// TwinCAT 3 PLC project PLC
// ProgramVersion: 3.1.4026.20
// libraries:
//   Tc2_Standard, * (Beckhoff Automation GmbH)
//   Tc2_System, * (Beckhoff Automation GmbH)
//   Tc2_Utilities, * (Beckhoff Automation GmbH)
//   Tc3_EventLogger, * (Beckhoff Automation GmbH)
// project tree:
//   DUTs/HMI/ ST_Batch_HMI.TcDUT, ST_Camera_HMI.TcDUT, ST_Counter_HMI.TcDUT, ST_Feeder_HMI.TcDUT, ST_Footer_HMI.TcDUT, ST_FromHMI.TcDUT, ST_Greasing_HMI.TcDUT, ST_History_HMI.TcDUT, ST_Lift_HMI.TcDUT, ST_MachineControl_HMI.TcDUT, ST_MachineInfo_HMI.TcDUT, ST_Navigation_HMI.TcDUT, ST_PID_HMI.TcDUT, ST_Robot_HMI.TcDUT, ST_Station_HMI.TcDUT, ST_ToHMI.TcDUT
//   DUTs/ ST_Alarm.TcDUT, ST_Batch.TcDUT, ST_Control.TcDUT, ST_Settings.TcDUT, ST_StationCommand.TcDUT
//   DUTs/Time/ ST_DateAndTime.TcDUT, ST_Time.TcDUT
//   DUTs/Trend/ ST_Point.TcDUT
//   FBs/Devices/ FB_Counter.TcPOU, FB_Device.TcPOU, FB_Greaser.TcPOU, FB_Handshake.TcPOU, FB_Stepper.TcPOU
//   FBs/ FB_AlarmDiagnostic.TcPOU, FB_Batch.TcPOU, FB_SystemDateTime.TcPOU, FB_TONP.TcPOU
//   Functions/ F_Message.TcPOU, F_StepCMP.TcPOU, F_TimerToString.TcPOU
//   GVLs/ CONST.TcGVL, GV.TcGVL, HMI.TcGVL, IN.TcGVL, OUT.TcGVL, Station.TcGVL
//   / PlcTask.TcTTO
//   POUs/ MAIN.TcPOU, P00_Mapping.TcPOU, P01_AnalogScaling.TcPOU, P02_GlobalSystemTime.TcPOU, P03_MachineControl.TcPOU, P05_DeviceControl.TcPOU, P06_ProcessControl.TcPOU, P99_HMIControl.TcPOU
//   POUs/Sequences/ Camera.TcPOU, Conveyor.TcPOU, Feeder.TcPOU, Greaser.TcPOU, IntakeBuffer.TcPOU, OutletBuffer.TcPOU, Robot.TcPOU
//   POUs/Simulation/ Service_sim.TcPOU, Simulation.TcPOU
// real-time tasks:
//   TASK PlcTask: cycle T#10ms, priority 20, ADS port 350

CONFIGURATION PLC
    RESOURCE PLC ON TwinCAT3
        TASK PlcTask(INTERVAL := T#10ms, PRIORITY := 20);
        PROGRAM MAIN WITH PlcTask : MAIN;
    END_RESOURCE
END_CONFIGURATION

// ---- DUTs/HMI/ST_Batch_HMI.TcDUT
TYPE ST_Batch_HMI :
STRUCT
	bBatchOpen : BOOL;
	bBatchClose : BOOL;
	sBatchName : STRING;
END_STRUCT
END_TYPE

// ---- DUTs/HMI/ST_Camera_HMI.TcDUT
TYPE ST_Camera_HMI :
STRUCT
	bCapturing		:BOOL;
	sCameraStatus	:STRING;
	sJobResult		:STRING;
END_STRUCT
END_TYPE

// ---- DUTs/HMI/ST_Counter_HMI.TcDUT
TYPE ST_Counter_HMI :
STRUCT
	bReset			:BOOL;
	iOK				:UDINT;
	iNOK			:UDINT;
	bError			:BOOL;
END_STRUCT
END_TYPE

// ---- DUTs/HMI/ST_Feeder_HMI.TcDUT
TYPE ST_Feeder_HMI :
STRUCT
	bActivate		:BOOL;
	bDeactivate		:BOOL;
END_STRUCT
END_TYPE

// ---- DUTs/HMI/ST_Footer_HMI.TcDUT
TYPE ST_Footer_HMI :
STRUCT
	bAuto : BOOL; 
	bService : BOOL;
	bStop : BOOL;
	bStart : BOOL;
	bPause : BOOL;
	
	bAuto_Enable : BOOL;
	bService_Enable : BOOL;
	bStop_Enable : BOOL;
	bStart_Enable : BOOL;
	bPause_Enable : BOOL;
END_STRUCT
END_TYPE

// ---- DUTs/HMI/ST_FromHMI.TcDUT
TYPE ST_FromHMI :
STRUCT
	stMachineCtrl		: ST_MachineControl_HMI; //Footer commands
	stNavigation		: ST_Navigation_HMI;
	stRobot				: ST_Robot_HMI;
	stLiftIntake		: ST_Lift_HMI;
	stLiftOutlet		: ST_Lift_HMI;
	bConveyorJog		: BOOL;
	bRobotCameraCapture	: BOOL;
	bFixedCameraCapture	: BOOL;
	stBatch				: ST_Batch_HMI;
	stCounter			:ARRAY [1..4] OF ST_Counter_HMI;
	stGreasing			: ST_Greasing_HMI;
	iSelectedTray		: USINT;
	stFeeder			:ST_Feeder_HMI;
END_STRUCT
END_TYPE

// ---- DUTs/HMI/ST_Greasing_HMI.TcDUT
TYPE ST_Greasing_HMI :
STRUCT
	bPurge		:BOOL;
	bPulse		:BOOL;
	iTime		:UINT;
END_STRUCT
END_TYPE

// ---- DUTs/HMI/ST_History_HMI.TcDUT
TYPE ST_History_HMI :
STRUCT
	iOK	:UDINT;
	iNOK :UDINT;
	bShift1	:BOOL;
	bShift2 :BOOL;
	bShift3 :BOOL;
END_STRUCT
END_TYPE

// ---- DUTs/HMI/ST_Lift_HMI.TcDUT
TYPE ST_Lift_HMI :
STRUCT
	bHome		:BOOL;
	bGoUp		:BOOL;
	bGoDown		:BOOL;
	iPosition	:UINT;
END_STRUCT
END_TYPE

// ---- DUTs/HMI/ST_MachineControl_HMI.TcDUT
TYPE ST_MachineControl_HMI :
STRUCT
	bAutomaticMode 		: BOOL;
	bServiceMode		: BOOL;
	
	bStartProcess		: BOOL;
	bPauseProcess		: BOOL;
	bStopProcess		: BOOL;
	
	
END_STRUCT
END_TYPE

// ---- DUTs/HMI/ST_MachineInfo_HMI.TcDUT
TYPE ST_MachineInfo_HMI :
STRUCT
	bControlMode		: BOOL;//0 - Auto, 1 - Manual
	iStatus				: USINT;//0-Stopping, 1-Stopped, 2-Starting, 3-Running, 4-Paused
	sBatch				: STRING;// Closed or Batch number
	iCounter			: LINT;//Finished part counter
	sDate				: STRING;//System date
	sTime				: STRING;//System time
	sCycleTime			: STRING;//MM:SS
	sUserLogged			: STRING;
	iCurrentStep		: USINT;
	
END_STRUCT
END_TYPE

// ---- DUTs/HMI/ST_Navigation_HMI.TcDUT
TYPE ST_Navigation_HMI :
STRUCT
	
END_STRUCT
END_TYPE

// ---- DUTs/HMI/ST_PID_HMI.TcDUT
TYPE ST_PID_HMI :
STRUCT
	bTray_PickPosition	: BOOL;
	bTray_PlacePosition	: BOOL;
	bTray_Ready_Left	: BOOL;
	bTray_Ready_Right	: BOOL;
	bConveyor_Moving	: BOOL;
END_STRUCT
END_TYPE

// ---- DUTs/HMI/ST_Robot_HMI.TcDUT
TYPE ST_Robot_HMI :
STRUCT
	bStart : BOOL;
	bStop : BOOL;
	bInit : BOOL;
	bPause	: BOOL;
	bPowerOn : BOOL;
	bPowerOff : BOOL;
	
	iStep : 	UINT;
	sStatus : STRING;
END_STRUCT
END_TYPE

// ---- DUTs/HMI/ST_Station_HMI.TcDUT
TYPE ST_Station_HMI :
STRUCT
	iStep			:UINT;
	bInterlocksOK	:BOOL;
	bReset			:BOOL;
	iStatus			:UINT;
END_STRUCT
END_TYPE

// ---- DUTs/HMI/ST_ToHMI.TcDUT
TYPE ST_ToHMI :
STRUCT
	stHeader		:ST_MachineInfo_HMI;
	stPID			:ST_PID_HMI;
	stFooter		:ST_Footer_HMI;
	stRobot			:ST_Robot_HMI;
	stLiftIntake	:ST_Lift_HMI;
	stLiftOutlet	:ST_Lift_HMI;
	bConveyorJog	:BOOL;
	stRobotCamera	:ST_Camera_HMI;
	stFixedCamera	:ST_Camera_HMI;
	stBatch			:ST_Batch_HMI;
	stCounter		:ARRAY [1..7] OF ST_Counter_HMI;
	stGreasing		:ST_Greasing_HMI;
	stHistory		:ST_History_HMI;
	iMessage		:UINT;
	iMessageSeverity :USINT;
	stFeeder		:ST_Feeder_HMI;
END_STRUCT
END_TYPE

// ---- DUTs/ST_Alarm.TcDUT
TYPE ST_Alarm :
STRUCT
	Alarm			:ARRAY[0..50] OF fb_TcAlarm;
	Active			:ARRAY[0..50] OF BOOL;
	Raise			:ARRAY[0..50] OF BOOL;
	
END_STRUCT
END_TYPE

// ---- DUTs/ST_Batch.TcDUT
TYPE ST_Batch :
STRUCT
	sBatchNumber		:STRING;
	sRecipeName			:STRING;
	sProductName		:STRING;
	sUser				:STRING;
	sStarted			:STRING;
	sFinished			:STRING;
END_STRUCT
END_TYPE

// ---- DUTs/ST_Control.TcDUT
TYPE ST_Control :
STRUCT
	iStep					:UINT;
	iStep_Prev				:UINT;
	bAuto					:BOOL;
	bService				:BOOL;
	bStarting				:BOOL;
	bInterlockOK			:BOOL;
	bProcesslockOK			:BOOL;
	bStartConditionsOK		:BOOL;
	bRunning				:BOOL;
	bPaused					:BOOL;
	bAbort					:BOOL;
	bStopping				:BOOL;
	bStopped				:BOOL;
	bJump					:BOOL;
	bHold					:BOOL;
	bPoweredOn				:BOOL;
	bPoweredOff				:BOOL;
	bInit					:BOOL;
END_STRUCT
END_TYPE

// ---- DUTs/ST_Settings.TcDUT
TYPE ST_Settings :
STRUCT
	//Timeout settings
	tCameraTimeout			:TIME;
	tConveyorTimeout		:TIME;
	tPickClampTimeout		:TIME;
	tPlaceClampTimeout		:TIME;
	tFeederTimeout			:TIME;
	tRobotTimeout			:TIME;
	
	//Process settings
	tGreasingPulseTime		:TIME;
END_STRUCT
END_TYPE

// ---- DUTs/ST_StationCommand.TcDUT
TYPE ST_StationCommand :
STRUCT
	//Feeder cmd
	bFeederSTART		:BOOL;
	//Intake lift cmd
	iIntakeLift_SP		:UINT;
	bIntakeLift_HOME	:BOOL;
	//Outlet lift cmd
	iOutletLift_SP		:UINT;
	bOutletLift_HOME	:BOOL;
	//Robot cmd
	bRobot_START		:BOOL;
	iRobot_JobNumber	:USINT;
	bRobot_Gripper		:BYTE;
	//Conveyor cmd
	bConveyorJog		:BOOL;
	bClampPick			:BOOL;
	bClampPlace			:BOOL;
	//Robot camera cmd
	bRobotCamera_Capture:BOOL;
	//Fixed camera cmd
	bFixedCamera_Capture:BOOL;
	iFixedCamera_Job	:USINT;
	//Counters
	bCount				:BOOL;
	iPartOK				:USINT;
	iPartNOK			:USINT;
	//Greasing
	bGreasing_Purge		:BOOL;
	bGreasing_Pulse		:BOOL;
	tGreasing_Time		:TIME;
END_STRUCT
END_TYPE

// ---- DUTs/Time/ST_DateAndTime.TcDUT
TYPE ST_DateAndTime :
STRUCT
END_STRUCT
END_TYPE

// ---- DUTs/Time/ST_Time.TcDUT
TYPE ST_Time :
STRUCT
	dtDateTime			:DT;
	sTime				:STRING;
	sDate				:STRING;
	sDateTime			:STRING;
	sFormatDateTime		:STRING;
	bClock_500ms		:BOOL;
	bClock_1s			:BOOL;
	bClock_2s			:BOOL;
	bClock_5s			:BOOL;
	bClock_60s			:BOOL;
	bClock_1OFF_2ON		:BOOL;
	bPulse_10s			:BOOL;
	bPulse_30s			:BOOL;
	bPulse_60s			:BOOL;
	bCustomBlink1		:BOOL;
	bCustomBlink2		:BOOL;
	bCustomBlink3		:BOOL;
	bNewHour			:BOOL;
	bNewDay				:BOOL;
	bNewMonth			:BOOL;
	bNewYear			:BOOL;
	CurrentHour			:WORD;
	CurrentDay			:WORD;
	CurrentMonth		:WORD;
	CurrentYear			:WORD;
END_STRUCT
END_TYPE

// ---- DUTs/Trend/ST_Point.TcDUT
TYPE ST_Point :
STRUCT
	x	:UDINT;
	y	:UDINT;
END_STRUCT
END_TYPE

// ---- GVLs/CONST.TcGVL
{attribute 'qualified_only'}
VAR_GLOBAL
	AMS_NETID				:STRING:='10.0.0.5.1.1';
	PROJECT_DIR				:STRING:='C:\250605-Aeromatic1\';
	DB_ID					:UDINT:=1;
	
	
	//Process constants
	GREASE_DENSITY			:REAL:=1;//[g/l]
	
	
	//Message IDs
	MSG_FillIntakeBuffer	:UINT := 10;
	
END_VAR

// ---- GVLs/GV.TcGVL
{attribute 'qualified_only'}
VAR_GLOBAL
	//Time
	stTime : ST_Time;
	bUPSDetect : BOOL;
END_VAR

VAR_GLOBAL PERSISTENT
	sUserLogged					:STRING;
	cntResettable				:FB_Counter;
	cntHourly					:FB_Counter;
	cntTotal					:FB_Counter;
	cntBatch					:FB_Counter;
	cntShift1					:FB_Counter;
	cntShift2					:FB_Counter;
	cntShift3					:FB_Counter;
	stSettings					:ST_Settings;
	aTrays						:ARRAY[1..10] OF ARRAY[1..14,1..7] OF BOOL;
END_VAR

// ---- GVLs/HMI.TcGVL
{attribute 'qualified_only'}
VAR_GLOBAL
	stToHMI 			:ST_ToHMI;
	stFromHMI 			:ST_FromHMI; 
	iMenu 				:USINT;
	iPopupMenu 			:USINT;
	stGreasing			:ST_Station_HMI;
	stInletBuffer		:ST_Station_HMI;
	stOutletBuffer		:ST_Station_HMI;
	stConveyor			:ST_Station_HMI;
	stRobot				:ST_Station_HMI;
	stCamera			:ST_Station_HMI;
	stFeeder			:ST_Station_HMI;
	stLastTray			:ARRAY[1..14,1..7] OF BOOL;
END_VAR

// ---- GVLs/IN.TcGVL
{attribute 'qualified_only'}
VAR_GLOBAL
	//Input modules:


	//Input variables:	
	
	//Sensors
	bSensor_TrayInReady		:BOOL;
	bSensor_TrayOutReady	:BOOL;
	bSensor_TrayInPick		:BOOL;
	bSensor_TrayInPlace		:BOOL;
	bSensor_InletDoor_Closed	:BOOL;
	bSensor_OutletDoor_Closed	:BOOL;
	
	//Robot
	bRobot_Initialised		:BOOL;
	bRobot_Running			:BOOL;
	bRobot_Ready			:BOOL;
	bRobot_On				:BOOL;
	bRobot_Ok				:BOOL;
	bRobot_Done				:BOOL;
	bRobot_Gripper			:BYTE;
	bRobot_Args				:BYTE;
	
	//Camera
	bCamera_Busy			:BOOL;
	bCamera_Done			:BOOL;
	bCamera_Args			:BYTE;
	bCamera_On				:BOOL;
	
	//Conveyor
	bConveyor_Drive			:BOOL;
	bPickClamped			:BOOL;
	bPlaceClamped			:BOOL;
	bConveyorDrive_OK		:BOOL;
	
	//Feeder
	bFeeder_ON				:BOOL;
	bFeederDrive_OK			:BOOL;
	
	//Intake buffer
	bIntakeBuffer_Homed		:BOOL;
	iBufferIn				:INT;
	bIntakeBuffer_DriveOK	:BOOL;
	//Outlet buffer
	bOutletBuffer_Homed		:BOOL;
	iBufferOut				:INT;
	bOutletBuffer_DriveOK	:BOOL;
	
	//Greaser
	bGreasing_PressureOK	:BOOL;
	bGreasing_LevelOK		:BOOL;

END_VAR

// ---- GVLs/OUT.TcGVL
{attribute 'qualified_only'}
VAR_GLOBAL
	//Camera
	bFixedCamera_Trigger		:BOOL;
	FixedCameraArgs				:ARRAY[0..9] OF BOOL;
	bFixedCamera_PlcReady		:BOOL;
	//Conveyor
	bConveyor_Jog				:BOOL;
	bClampPick					:BOOL;
	bClampPlace					:BOOL;
	//Robot
	bRobot_Execute				:BOOL;
	bRobot_PlcReady				:BOOL;
END_VAR

// ---- GVLs/Station.TcGVL
{attribute 'qualified_only'}
VAR_GLOBAL
	stAlarm							:ST_Alarm;

	bBatchOpen						:BOOL;
	bBatchClosed						:BOOL;
	bBatchBusy						:BOOL;
	bAlarmOK						:BOOL;	
	
	stAutoCmd						:ST_StationCommand;
	stManCmd						:ST_StationCommand;
	stCommand						:ST_StationCommand;				

	tonCycleTimer					:TON;

END_VAR

VAR_GLOBAL PERSISTENT
	stSettings						:ST_Settings;
	stBatch							:ST_Batch;
	stLastBatch						:ST_Batch;
	stControl						:ST_Control;
	stRobotControl					:ST_Control;
	
	iIntakeLiftPosition				:USINT;
	iOutletLiftPosition				:USINT;
END_VAR

// ---- POUs/MAIN.TcPOU
PROGRAM MAIN
VAR
	bFirstCycle		: BOOL := TRUE;
END_VAR



P02_GlobalSystemTime();
P03_MachineControl();
P03_MachineControl.Robot();
P03_MachineControl.Batch();
P05_DeviceControl();
P06_ProcessControl();
P99_HMIControl();

//Simulations
Service_sim();



bFirstCycle := FALSE;

END_PROGRAM

// ---- POUs/P02_GlobalSystemTime.TcPOU
PROGRAM P02_GlobalSystemTime
VAR
	fbGlobalTime 		:FB_SystemDateTIme;
END_VAR

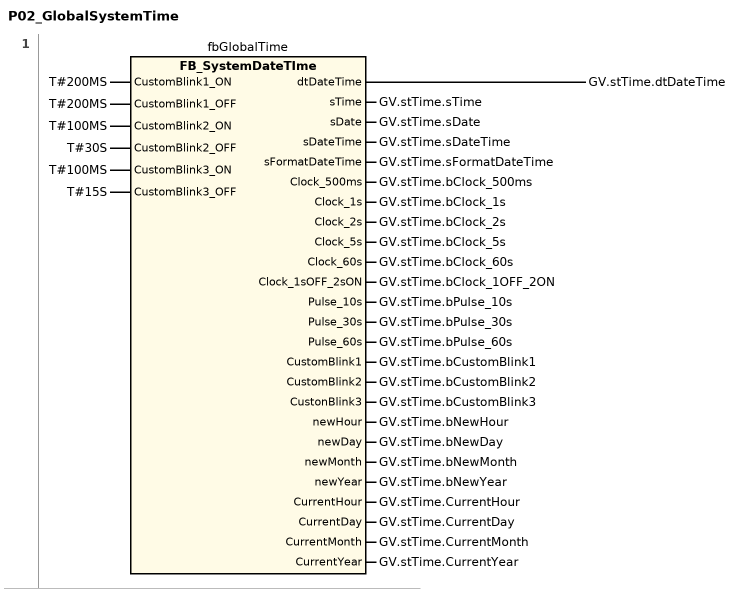
// NETWORK 1
fbGlobalTime(
    CustomBlink1_ON := T#200MS,
    CustomBlink1_OFF := T#200MS,
    CustomBlink2_ON := T#100MS,
    CustomBlink2_OFF := T#30S,
    CustomBlink3_ON := T#100MS,
    CustomBlink3_OFF := T#15S,
    sTime => GV.stTime.sTime,
    sDate => GV.stTime.sDate,
    sDateTime => GV.stTime.sDateTime,
    sFormatDateTime => GV.stTime.sFormatDateTime,
    Clock_500ms => GV.stTime.bClock_500ms,
    Clock_1s => GV.stTime.bClock_1s,
    Clock_2s => GV.stTime.bClock_2s,
    Clock_5s => GV.stTime.bClock_5s,
    Clock_60s => GV.stTime.bClock_60s,
    Clock_1sOFF_2sON => GV.stTime.bClock_1OFF_2ON,
    Pulse_10s => GV.stTime.bPulse_10s,
    Pulse_30s => GV.stTime.bPulse_30s,
    Pulse_60s => GV.stTime.bPulse_60s,
    CustomBlink1 => GV.stTime.bCustomBlink1,
    CustomBlink2 => GV.stTime.bCustomBlink2,
    CustonBlink3 => GV.stTime.bCustomBlink3,
    newHour => GV.stTime.bNewHour,
    newDay => GV.stTime.bNewDay,
    newMonth => GV.stTime.bNewMonth,
    newYear => GV.stTime.bNewYear,
    CurrentHour => GV.stTime.CurrentHour,
    CurrentDay => GV.stTime.CurrentDay,
    CurrentMonth => GV.stTime.CurrentMonth,
    CurrentYear => GV.stTime.CurrentYear); // FB_SystemDateTIme
GV.stTime.dtDateTime := fbGlobalTime.dtDateTime;

END_PROGRAM

// ---- FBs/FB_SystemDateTime.TcPOU
// Created by Dimitar Stojanov 06.2023 
// Install TC2_Utilities and Import ST_Time structure for fully functionality of this block


FUNCTION_BLOCK FB_SystemDateTime
VAR_INPUT
	CustomBlink1_ON		:TIME;
	CustomBlink1_OFF	:TIME;
	CustomBlink2_ON		:TIME;
	CustomBlink2_OFF	:TIME;
	CustomBlink3_ON		:TIME;
	CustomBlink3_OFF	:TIME;
END_VAR
VAR_OUTPUT
	dtDateTime		:DT;
	sTime			:STRING;
	sDate			:STRING;
	sDateTime		:STRING;
	sFormatDateTime	:STRING;
	Clock_500ms		:BOOL;
	Clock_1s		:BOOL;
	Clock_2s		:BOOL;
	Clock_5s		:BOOL;
	Clock_60s		:BOOL;
	Clock_1sOFF_2sON	:BOOL;
	Pulse_10s		:BOOL;
	Pulse_30s		:BOOL;
	Pulse_60s		:BOOL;
	CustomBlink1	:BOOL;
	CustomBlink2	:BOOL;
	CustonBlink3	:BOOL;
	newHour			:BOOL; //true for 1 cycle when hour change
	newDay			:BOOL;
	newMonth		:BOOL;
	newYear			:BOOL;
END_VAR
VAR
	bFirstCycle		:BOOL:=TRUE;	

	fbTime			:FB_LocalSystemTime;
	systemDateTime	:TIMESTRUCT;
	
	Second			:STRING;
	Minute			:STRING;
	Hour			:STRING;
	Day				:STRING;
	Month			:STRING;
	Year			:STRING;
	
	iClock1s		:INT;
	TON_0: TON;
	TOF_0: TOF;
	TON_1: TON;
	TOF_1: TOF;
	TOF_2: TOF;
	TON_2: TON;
	TON_3: TON;
	TOF_3: TOF;
	TOF_4: TOF;
	TON_4: TON;
	TON_5: TON;
	TOF_5: TOF;
	TON_6: TON;
	TOF_6: TOF;
	TON_7: TON;
	TOF_7: TOF;
	TON_8: TON;
	TOF_8: TOF;
	
	TON_9: TON;
	TOF_9: TOF;
	TOF_10: TOF;
	TOF_11: TOF;
	TON_10: TON;
	TON_20: TON;
	TOF_20: TOF;
	TON_21: TON;
	TOF_21: TOF;
	TON_22: TON;
	TOF_22: TOF;
	
	TOF_23: TOF;
	
	bDelay			:BOOL;
	TON_DELAY		:TON;
END_VAR

VAR_OUTPUT PERSISTENT
	CurrentHour		:WORD;
	CurrentDay		:WORD;
	CurrentMonth	:WORD;
	CurrentYear		:WORD;
END_VAR

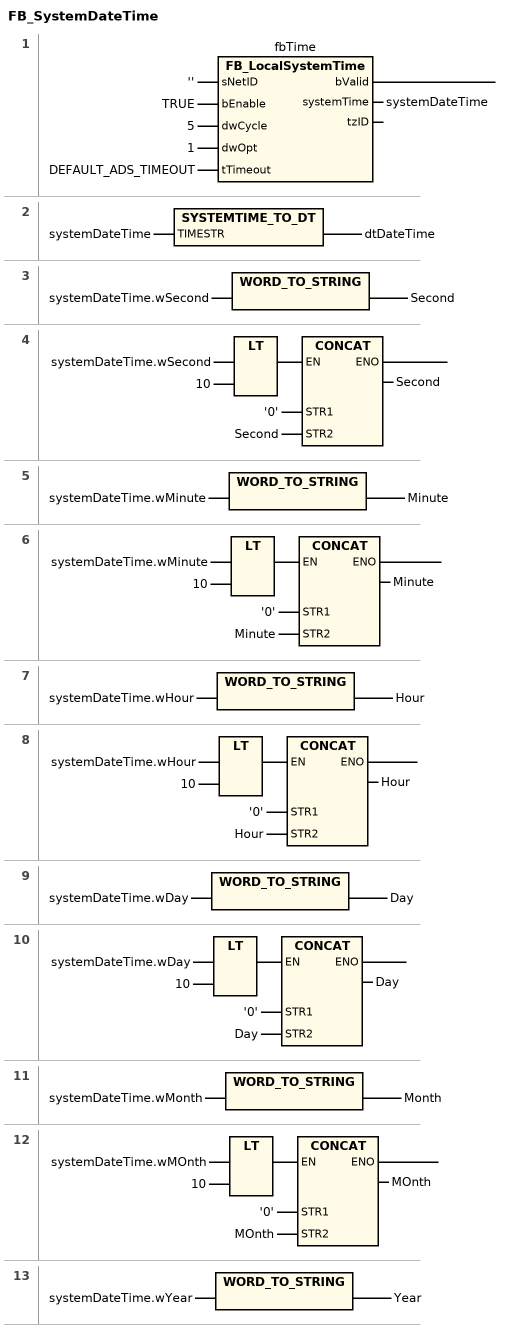
// NETWORK 1
fbTime(
    sNetID := '',
    bEnable := TRUE,
    dwCycle := 5,
    dwOpt := 1,
    tTimeout := DEFAULT_ADS_TIMEOUT,
    systemTime => systemDateTime); // FB_LocalSystemTime

// NETWORK 2
dtDateTime := SYSTEMTIME_TO_DT(TIMESTR := systemDateTime);

// NETWORK 3
Second := WORD_TO_STRING(systemDateTime.wSecond);

// NETWORK 4
IF systemDateTime.wSecond < 10 THEN Second := CONCAT(STR1 := '0', STR2 := Second); END_IF

// NETWORK 5
Minute := WORD_TO_STRING(systemDateTime.wMinute);

// NETWORK 6
IF systemDateTime.wMinute < 10 THEN Minute := CONCAT(STR1 := '0', STR2 := Minute); END_IF

// NETWORK 7
Hour := WORD_TO_STRING(systemDateTime.wHour);

// NETWORK 8
IF systemDateTime.wHour < 10 THEN Hour := CONCAT(STR1 := '0', STR2 := Hour); END_IF

// NETWORK 9
Day := WORD_TO_STRING(systemDateTime.wDay);

// NETWORK 10
IF systemDateTime.wDay < 10 THEN Day := CONCAT(STR1 := '0', STR2 := Day); END_IF

// NETWORK 11
Month := WORD_TO_STRING(systemDateTime.wMonth);

// NETWORK 12
IF systemDateTime.wMOnth < 10 THEN MOnth := CONCAT(STR1 := '0', STR2 := MOnth); END_IF

// NETWORK 13
Year := WORD_TO_STRING(systemDateTime.wYear);

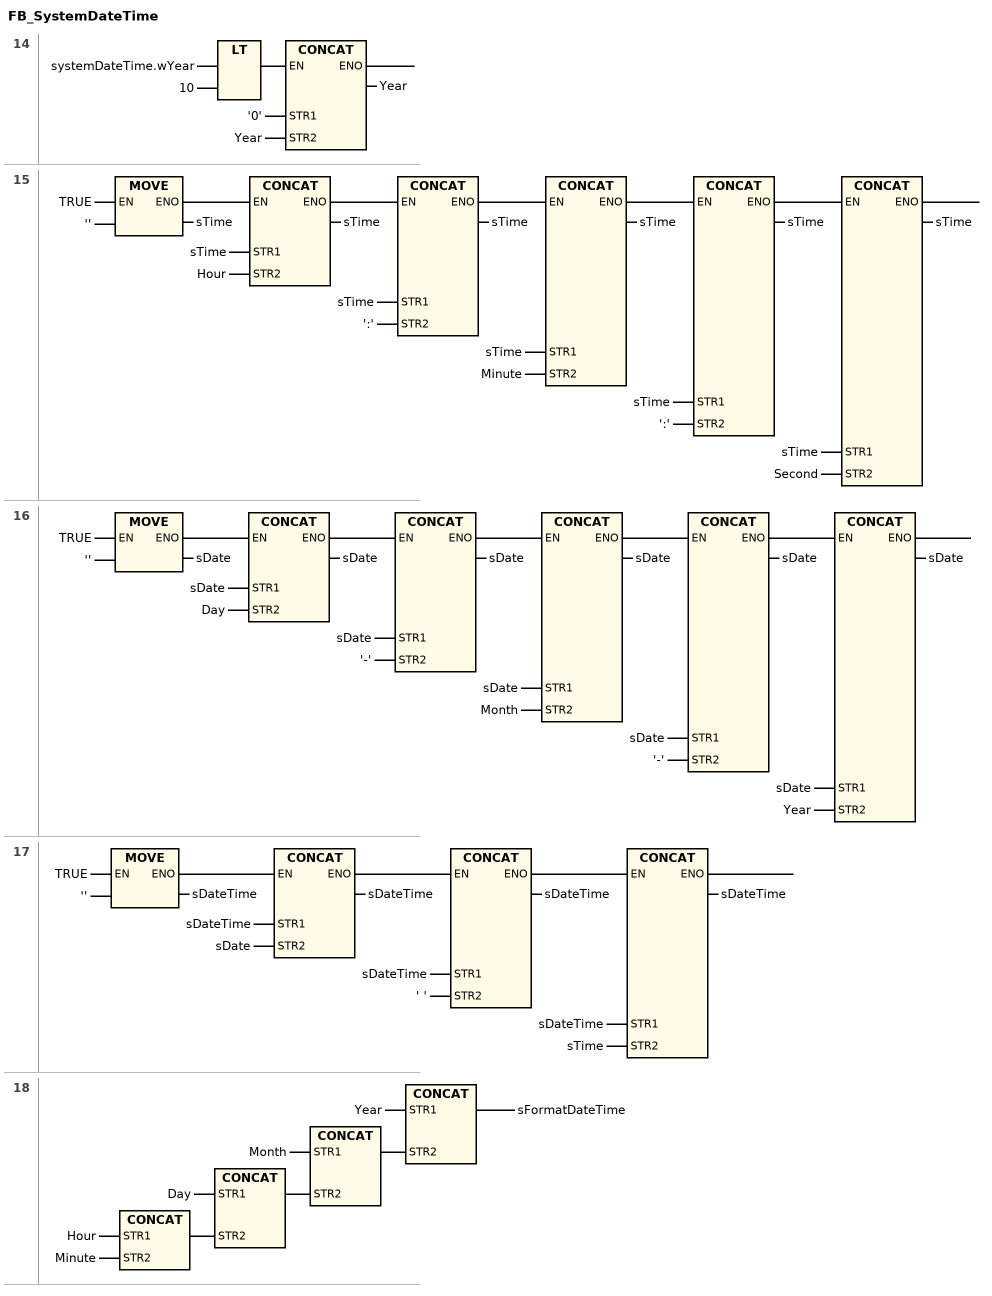
// NETWORK 14
IF systemDateTime.wYear < 10 THEN Year := CONCAT(STR1 := '0', STR2 := Year); END_IF

// NETWORK 15
sTime := '';
sTime := CONCAT(STR1 := sTime, STR2 := Hour);
sTime := CONCAT(STR1 := sTime, STR2 := ':');
sTime := CONCAT(STR1 := sTime, STR2 := Minute);
sTime := CONCAT(STR1 := sTime, STR2 := ':');
sTime := CONCAT(STR1 := sTime, STR2 := Second);

// NETWORK 16
sDate := '';
sDate := CONCAT(STR1 := sDate, STR2 := Day);
sDate := CONCAT(STR1 := sDate, STR2 := '-');
sDate := CONCAT(STR1 := sDate, STR2 := Month);
sDate := CONCAT(STR1 := sDate, STR2 := '-');
sDate := CONCAT(STR1 := sDate, STR2 := Year);

// NETWORK 17
sDateTime := '';
sDateTime := CONCAT(STR1 := sDateTime, STR2 := sDate);
sDateTime := CONCAT(STR1 := sDateTime, STR2 := ' ');
sDateTime := CONCAT(STR1 := sDateTime, STR2 := sTime);

// NETWORK 18
sFormatDateTime := CONCAT(STR1 := Year, STR2 := CONCAT(STR1 := Month, STR2 := CONCAT(STR1 := Day, STR2 := CONCAT(STR1 := Hour, STR2 := Minute))));

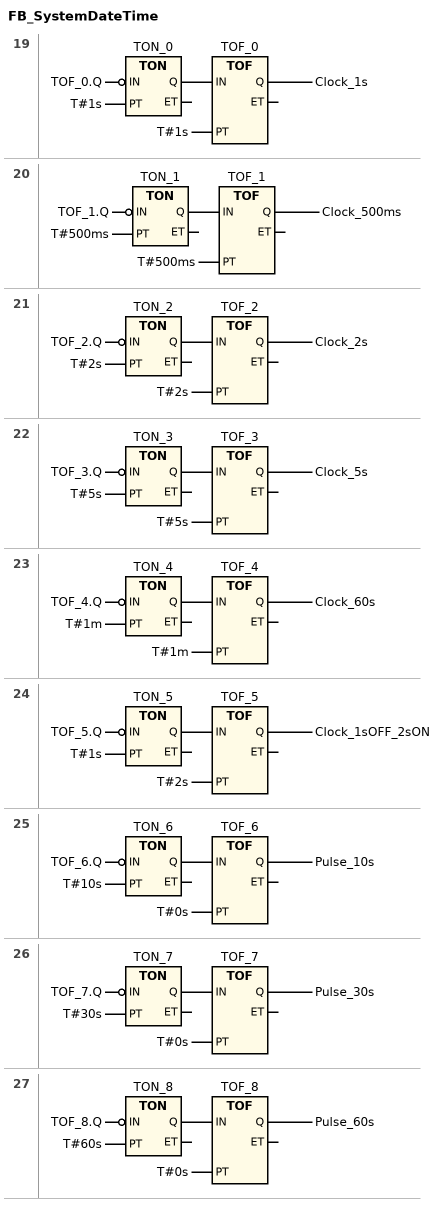
// NETWORK 19
TON_0(IN := NOT TOF_0.Q, PT := T#1s); // TON
TOF_0(IN := TON_0.Q, PT := T#1s); // TOF
Clock_1s := TOF_0.Q;

// NETWORK 20
TON_1(IN := NOT TOF_1.Q, PT := T#500ms); // TON
TOF_1(IN := TON_1.Q, PT := T#500ms); // TOF
Clock_500ms := TOF_1.Q;

// NETWORK 21
TON_2(IN := NOT TOF_2.Q, PT := T#2s); // TON
TOF_2(IN := TON_2.Q, PT := T#2s); // TOF
Clock_2s := TOF_2.Q;

// NETWORK 22
TON_3(IN := NOT TOF_3.Q, PT := T#5s); // TON
TOF_3(IN := TON_3.Q, PT := T#5s); // TOF
Clock_5s := TOF_3.Q;

// NETWORK 23
TON_4(IN := NOT TOF_4.Q, PT := T#1m); // TON
TOF_4(IN := TON_4.Q, PT := T#1m); // TOF
Clock_60s := TOF_4.Q;

// NETWORK 24
TON_5(IN := NOT TOF_5.Q, PT := T#1s); // TON
TOF_5(IN := TON_5.Q, PT := T#2s); // TOF
Clock_1sOFF_2sON := TOF_5.Q;

// NETWORK 25
TON_6(IN := NOT TOF_6.Q, PT := T#10s); // TON
TOF_6(IN := TON_6.Q, PT := T#0s); // TOF
Pulse_10s := TOF_6.Q;

// NETWORK 26
TON_7(IN := NOT TOF_7.Q, PT := T#30s); // TON
TOF_7(IN := TON_7.Q, PT := T#0s); // TOF
Pulse_30s := TOF_7.Q;

// NETWORK 27
TON_8(IN := NOT TOF_8.Q, PT := T#60s); // TON
TOF_8(IN := TON_8.Q, PT := T#0s); // TOF
Pulse_60s := TOF_8.Q;

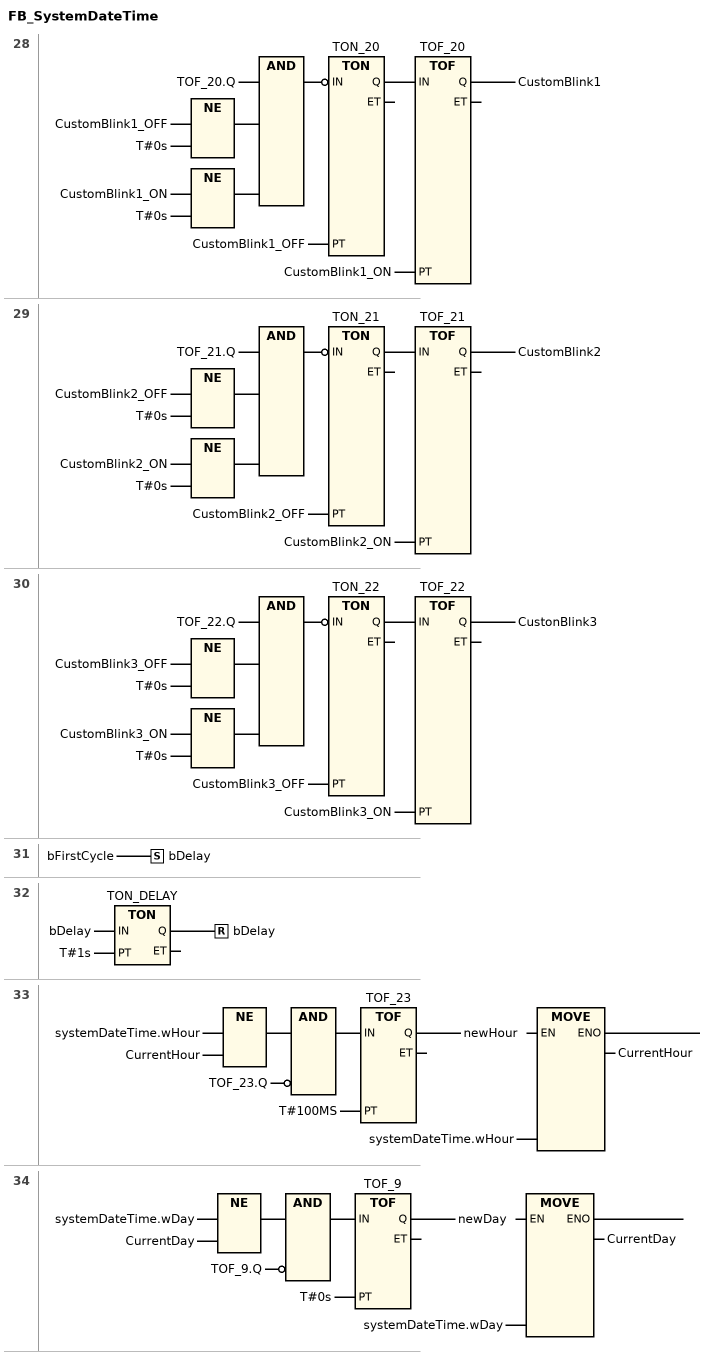
// NETWORK 28
TON_20(IN := NOT (TOF_20.Q AND CustomBlink1_OFF <> T#0s AND CustomBlink1_ON <> T#0s), PT := CustomBlink1_OFF); // TON
TOF_20(IN := TON_20.Q, PT := CustomBlink1_ON); // TOF
CustomBlink1 := TOF_20.Q;

// NETWORK 29
TON_21(IN := NOT (TOF_21.Q AND CustomBlink2_OFF <> T#0s AND CustomBlink2_ON <> T#0s), PT := CustomBlink2_OFF); // TON
TOF_21(IN := TON_21.Q, PT := CustomBlink2_ON); // TOF
CustomBlink2 := TOF_21.Q;

// NETWORK 30
TON_22(IN := NOT (TOF_22.Q AND CustomBlink3_OFF <> T#0s AND CustomBlink3_ON <> T#0s), PT := CustomBlink3_OFF); // TON
TOF_22(IN := TON_22.Q, PT := CustomBlink3_ON); // TOF
CustonBlink3 := TOF_22.Q;

// NETWORK 31
bDelay S= bFirstCycle;

// NETWORK 32
TON_DELAY(IN := bDelay, PT := T#1s); // TON
bDelay R= TON_DELAY.Q;

// NETWORK 33
TOF_23(IN := systemDateTime.wHour <> CurrentHour AND NOT TOF_23.Q, PT := T#100MS); // TOF
newHour := TOF_23.Q;
IF TOF_23.Q THEN CurrentHour := systemDateTime.wHour; END_IF

// NETWORK 34
TOF_9(IN := systemDateTime.wDay <> CurrentDay AND NOT TOF_9.Q, PT := T#0s); // TOF
newDay := TOF_9.Q;
IF TOF_9.Q THEN CurrentDay := systemDateTime.wDay; END_IF

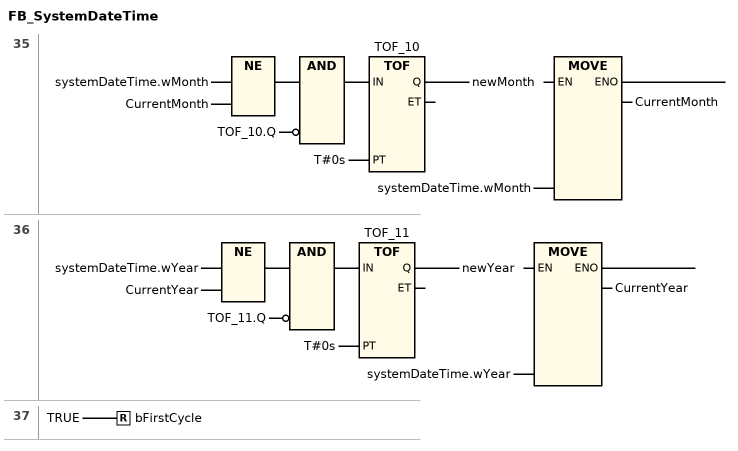
// NETWORK 35
TOF_10(IN := systemDateTime.wMonth <> CurrentMonth AND NOT TOF_10.Q, PT := T#0s); // TOF
newMonth := TOF_10.Q;
IF TOF_10.Q THEN CurrentMonth := systemDateTime.wMonth; END_IF

// NETWORK 36
TOF_11(IN := systemDateTime.wYear <> CurrentYear AND NOT TOF_11.Q, PT := T#0s); // TOF
newYear := TOF_11.Q;
IF TOF_11.Q THEN CurrentYear := systemDateTime.wYear; END_IF

// NETWORK 37
bFirstCycle R= TRUE;

END_FUNCTION_BLOCK

// ---- POUs/P03_MachineControl.TcPOU
PROGRAM P03_MachineControl
VAR
	tonStarting					:TON;
	tonStopping					:TON;
	tonRobotStarting			:TON;
	tonRobotStopping			:TON;
	tonRobotInitialising		:TON;
	
	bStop						:BOOL;
	
	fbBatch						:FB_Batch;
	tonBatchTime				:FB_TONP;
END_VAR
VAR // added by the converter: edge detectors and wires of the graphical bodies
    _w1, _w2, _w3, _w4, _w5, _w6, _w7, _w8, _w9, _w10, _w11, _w12 : BOOL;
    _rt1 : R_TRIG;
END_VAR

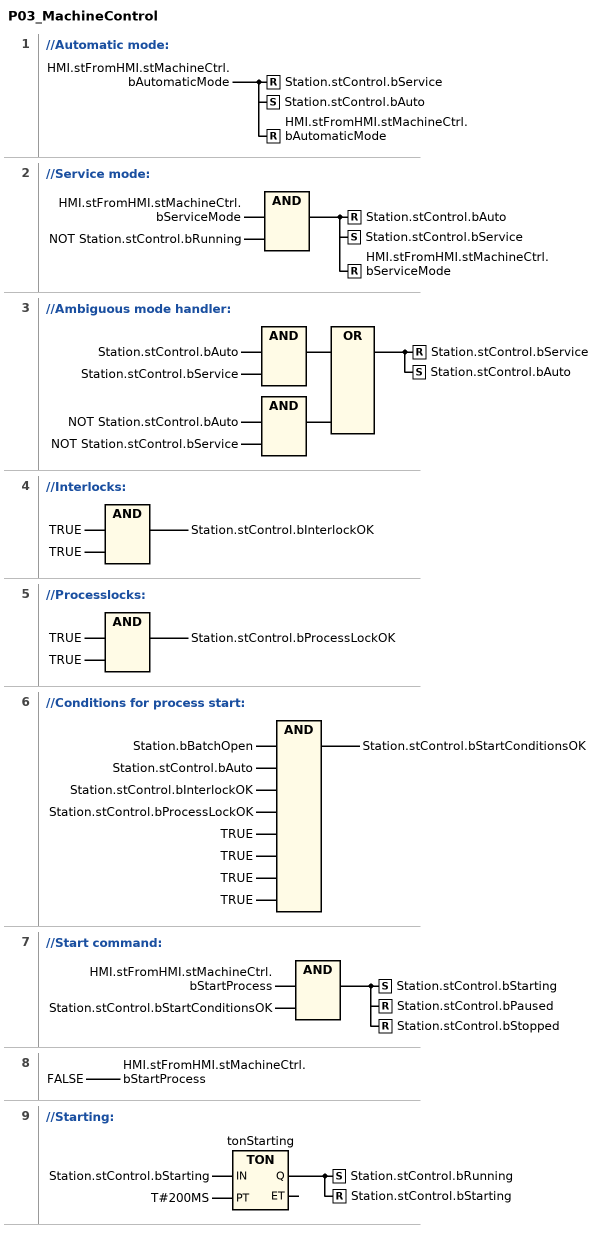
// NETWORK 1
// label: //Automatic mode
Station.stControl.bService R= HMI.stFromHMI.stMachineCtrl.bAutomaticMode;
Station.stControl.bAuto S= HMI.stFromHMI.stMachineCtrl.bAutomaticMode;
HMI.stFromHMI.stMachineCtrl.bAutomaticMode R= HMI.stFromHMI.stMachineCtrl.bAutomaticMode;

// NETWORK 2
// label: //Service mode
_w1 := HMI.stFromHMI.stMachineCtrl.bServiceMode AND (NOT Station.stControl.bRunning);
Station.stControl.bAuto R= _w1;
Station.stControl.bService S= _w1;
HMI.stFromHMI.stMachineCtrl.bServiceMode R= _w1;

// NETWORK 3
// label: //Ambiguous mode handler
_w2 := Station.stControl.bAuto AND Station.stControl.bService OR (NOT Station.stControl.bAuto) AND (NOT Station.stControl.bService);
Station.stControl.bService R= _w2;
Station.stControl.bAuto S= _w2;

// NETWORK 4
// label: //Interlocks
Station.stControl.bInterlockOK := TRUE AND TRUE;

// NETWORK 5
// label: //Processlocks
Station.stControl.bProcessLockOK := TRUE AND TRUE;

// NETWORK 6
// label: //Conditions for process start
Station.stControl.bStartConditionsOK := Station.bBatchOpen AND Station.stControl.bAuto AND Station.stControl.bInterlockOK AND Station.stControl.bProcessLockOK AND TRUE AND TRUE AND TRUE AND TRUE;

// NETWORK 7
// label: //Start command
_w3 := HMI.stFromHMI.stMachineCtrl.bStartProcess AND Station.stControl.bStartConditionsOK;
Station.stControl.bStarting S= _w3;
Station.stControl.bPaused R= _w3;
Station.stControl.bStopped R= _w3;

// NETWORK 8
HMI.stFromHMI.stMachineCtrl.bStartProcess := FALSE;

// NETWORK 9
// label: //Starting
tonStarting(IN := Station.stControl.bStarting, PT := T#200MS); // TON
Station.stControl.bRunning S= tonStarting.Q;
Station.stControl.bStarting R= tonStarting.Q;

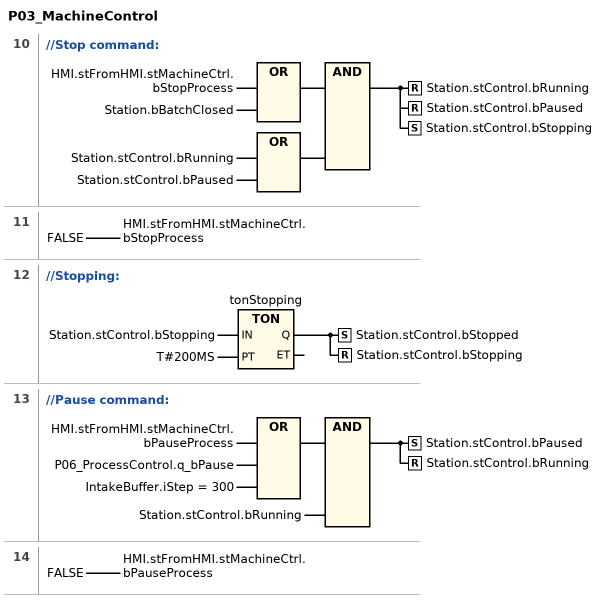
// NETWORK 10
// label: //Stop command
_w4 := (HMI.stFromHMI.stMachineCtrl.bStopProcess OR Station.bBatchClosed) AND (Station.stControl.bRunning OR Station.stControl.bPaused);
Station.stControl.bRunning R= _w4;
Station.stControl.bPaused R= _w4;
Station.stControl.bStopping S= _w4;

// NETWORK 11
HMI.stFromHMI.stMachineCtrl.bStopProcess := FALSE;

// NETWORK 12
// label: //Stopping
tonStopping(IN := Station.stControl.bStopping, PT := T#200MS); // TON
Station.stControl.bStopped S= tonStopping.Q;
Station.stControl.bStopping R= tonStopping.Q;

// NETWORK 13
// label: //Pause command
_w5 := (HMI.stFromHMI.stMachineCtrl.bPauseProcess OR P06_ProcessControl.q_bPause OR (IntakeBuffer.iStep = 300)) AND Station.stControl.bRunning;
Station.stControl.bPaused S= _w5;
Station.stControl.bRunning R= _w5;

// NETWORK 14
HMI.stFromHMI.stMachineCtrl.bPauseProcess := FALSE;

ACTION Batch:
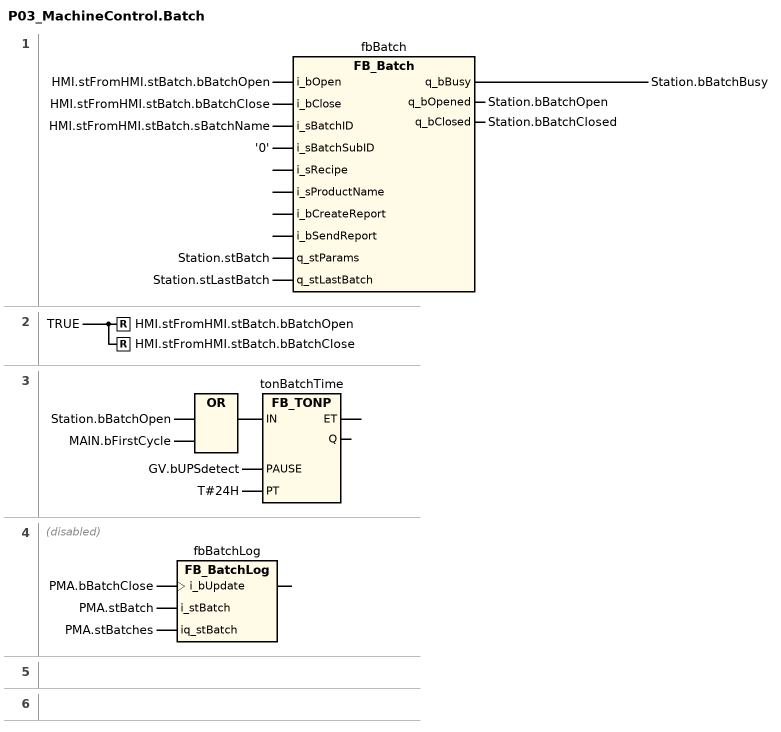
// NETWORK 1
fbBatch(
    i_bOpen := HMI.stFromHMI.stBatch.bBatchOpen,
    i_bClose := HMI.stFromHMI.stBatch.bBatchClose,
    i_sBatchID := HMI.stFromHMI.stBatch.sBatchName,
    i_sBatchSubID := '0',
    q_stParams := Station.stBatch,
    q_stLastBatch := Station.stLastBatch,
    q_bOpened => Station.bBatchOpen,
    q_bClosed => Station.bBatchClosed); // FB_Batch
Station.bBatchBusy := fbBatch.q_bBusy;

// NETWORK 2
HMI.stFromHMI.stBatch.bBatchOpen R= TRUE;
HMI.stFromHMI.stBatch.bBatchClose R= TRUE;

// NETWORK 3
tonBatchTime(IN := Station.bBatchOpen OR MAIN.bFirstCycle, PAUSE := GV.bUPSdetect, PT := T#24H); // FB_TONP

// NETWORK 4 (disabled)
// _rt1(CLK := PMA.bBatchClose);
// fbBatchLog(i_bUpdate := _rt1.Q, i_stBatch := PMA.stBatch, iq_stBatch := PMA.stBatches); // FB_BatchLog

// NETWORK 5

// NETWORK 6
END_ACTION

ACTION Robot:
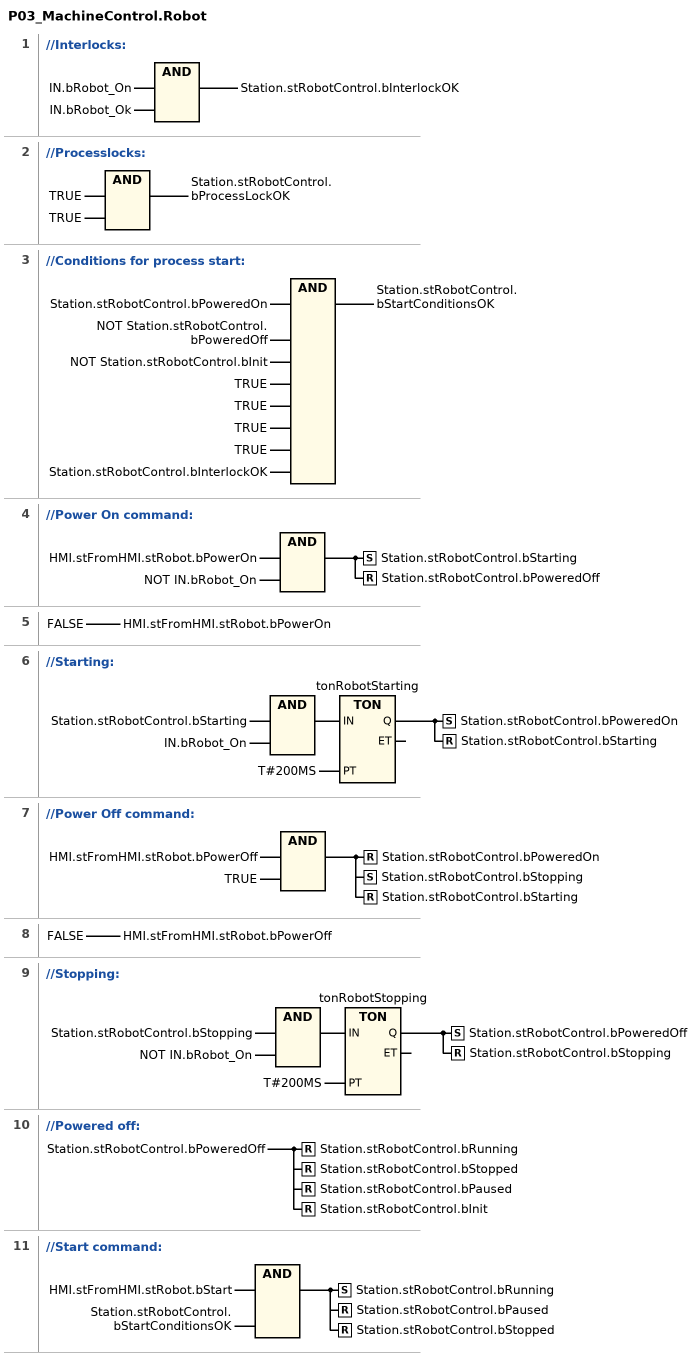
// NETWORK 1
// label: //Interlocks
Station.stRobotControl.bInterlockOK := IN.bRobot_On AND IN.bRobot_Ok;

// NETWORK 2
// label: //Processlocks
Station.stRobotControl.bProcessLockOK := TRUE AND TRUE;

// NETWORK 3
// label: //Conditions for process start
Station.stRobotControl.bStartConditionsOK := Station.stRobotControl.bPoweredOn AND (NOT Station.stRobotControl.bPoweredOff) AND (NOT Station.stRobotControl.bInit) AND TRUE AND TRUE AND TRUE AND TRUE AND Station.stRobotControl.bInterlockOK;

// NETWORK 4
// label: //Power On command
_w6 := HMI.stFromHMI.stRobot.bPowerOn AND (NOT IN.bRobot_On);
Station.stRobotControl.bStarting S= _w6;
Station.stRobotControl.bPoweredOff R= _w6;

// NETWORK 5
HMI.stFromHMI.stRobot.bPowerOn := FALSE;

// NETWORK 6
// label: //Starting
tonRobotStarting(IN := Station.stRobotControl.bStarting AND IN.bRobot_On, PT := T#200MS); // TON
Station.stRobotControl.bPoweredOn S= tonRobotStarting.Q;
Station.stRobotControl.bStarting R= tonRobotStarting.Q;

// NETWORK 7
// label: //Power Off command
_w7 := HMI.stFromHMI.stRobot.bPowerOff AND TRUE;
Station.stRobotControl.bPoweredOn R= _w7;
Station.stRobotControl.bStopping S= _w7;
Station.stRobotControl.bStarting R= _w7;

// NETWORK 8
HMI.stFromHMI.stRobot.bPowerOff := FALSE;

// NETWORK 9
// label: //Stopping
tonRobotStopping(IN := Station.stRobotControl.bStopping AND (NOT IN.bRobot_On), PT := T#200MS); // TON
Station.stRobotControl.bPoweredOff S= tonRobotStopping.Q;
Station.stRobotControl.bStopping R= tonRobotStopping.Q;

// NETWORK 10
// label: //Powered off
_w8 := Station.stRobotControl.bPoweredOff;
Station.stRobotControl.bRunning R= _w8;
Station.stRobotControl.bStopped R= _w8;
Station.stRobotControl.bPaused R= _w8;
Station.stRobotControl.bInit R= _w8;

// NETWORK 11
// label: //Start command
_w9 := HMI.stFromHMI.stRobot.bStart AND Station.stRobotControl.bStartConditionsOK;
Station.stRobotControl.bRunning S= _w9;
Station.stRobotControl.bPaused R= _w9;
Station.stRobotControl.bStopped R= _w9;

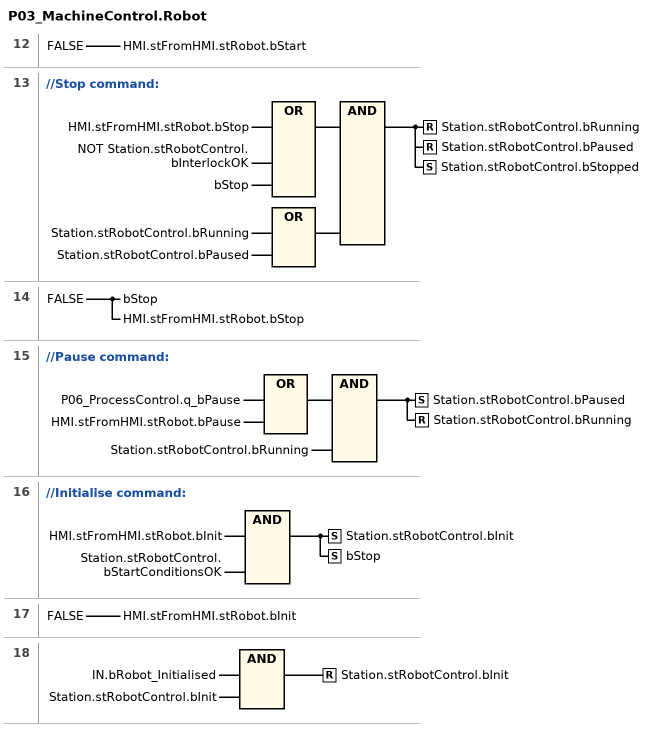
// NETWORK 12
HMI.stFromHMI.stRobot.bStart := FALSE;

// NETWORK 13
// label: //Stop command
_w10 := (HMI.stFromHMI.stRobot.bStop OR (NOT Station.stRobotControl.bInterlockOK) OR bStop) AND (Station.stRobotControl.bRunning OR Station.stRobotControl.bPaused);
Station.stRobotControl.bRunning R= _w10;
Station.stRobotControl.bPaused R= _w10;
Station.stRobotControl.bStopped S= _w10;

// NETWORK 14
bStop := FALSE;
HMI.stFromHMI.stRobot.bStop := FALSE;

// NETWORK 15
// label: //Pause command
_w11 := (P06_ProcessControl.q_bPause OR HMI.stFromHMI.stRobot.bPause) AND Station.stRobotControl.bRunning;
Station.stRobotControl.bPaused S= _w11;
Station.stRobotControl.bRunning R= _w11;

// NETWORK 16
// label: //Initialise command
_w12 := HMI.stFromHMI.stRobot.bInit AND Station.stRobotControl.bStartConditionsOK;
Station.stRobotControl.bInit S= _w12;
bStop S= _w12;

// NETWORK 17
HMI.stFromHMI.stRobot.bInit := FALSE;

// NETWORK 18
Station.stRobotControl.bInit R= IN.bRobot_Initialised AND Station.stRobotControl.bInit;
END_ACTION

END_PROGRAM

// ---- FBs/FB_Batch.TcPOU
FUNCTION_BLOCK FB_Batch
VAR_INPUT
	i_bOpen						:BOOL; 
	i_bClose					:BOOL; 
	i_sBatchID					:STRING; 
	i_sBatchSubID				:STRING;
	i_sRecipe					:STRING;
	i_sProductName				:STRING;
	i_bCreateReport				:BOOL;
	i_bSendReport				:BOOL;
END_VAR
VAR_IN_OUT
	q_stParams					:ST_Batch;
	q_stLastBatch				:ST_Batch;
END_VAR
VAR_OUTPUT
	q_bBusy						:BOOL;	
	q_bOpened					:BOOL:=FALSE; 
	q_bClosed					:BOOL:=FALSE; 		
END_VAR

VAR
	tDelayCreateReport			:TON;
	tDelaySendReport			:TON;
END_VAR	

VAR PERSISTENT
	iStep						:INT;
	sUserOpened					:STRING;
END_VAR

tDelayCreateReport(IN:=(iStep=200),PT:=T#3S);
tDelaySendReport(IN:=(iStep=300),PT:=T#3S);

CASE iStep OF

	0: 
		MEMSET(ADR(q_stParams),0,SIZEOF(q_stParams));
		IF i_bOpen THEN
			iStep:=50;
		END_IF
		
	50:
		IF i_sBatchSubID <> '0' THEN
			q_stParams.sBatchNumber:=CONCAT(i_sBatchID,'-');
			q_stParams.sBatchNumber:=CONCAT(q_stParams.sBatchNumber,i_sBatchSubID);
		ELSE
			q_stParams.sBatchNumber:=i_sBatchID;
		END_IF
		q_stParams.sRecipeName:=i_sRecipe;
		q_stParams.sProductName:=i_sProductName;
		q_stParams.sUser:=GV.sUserLogged;
		q_stParams.sStarted:=GV.stTime.sDateTime;
		sUserOpened:=GV.sUserLogged;
		iStep:=100;
			
	100:
		q_stParams.sUser:=sUserOpened;
		IF i_bClose THEN
			q_stParams.sFinished:=GV.stTime.sDateTime;
			q_stLastBatch:=q_stParams;
			iStep:=200;
		END_IF
		
	200:
		IF tDelayCreateReport.Q AND NOT i_bCreateReport THEN
			iStep:=300;
		END_IF
	300:
		IF tDelaySendReport.Q AND NOT i_bSendReport THEN
			iStep:=1000;
		END_IF
		
	1000:
		iStep:=0;	
END_CASE

q_bBusy:=iStep<>0;
q_bOpened:=iStep=100;
q_bClosed:=iStep>100;

END_FUNCTION_BLOCK

// ---- FBs/FB_TONP.TcPOU
FUNCTION_BLOCK FB_TONP
VAR_INPUT
	IN				:BOOL;
	PAUSE			:BOOL;
	PT				:TIME;
END_VAR
	
VAR_OUTPUT
	ET				:TIME;
	Q				:BOOL;
END_VAR
VAR
	TON				:TON;
	trigPause		:R_TRIG;
	trigStart		:R_TRIG;
	PT_START		:TIME;
	ET_PAUSE		:TIME;
END_VAR

trigStart(CLK:=IN);
trigPause(CLK:=PAUSE);

PT_START:=PT;
IF trigStart.Q THEN
	ET_PAUSE:=T#0S;
END_IF
IF IN AND trigPause.Q THEN
	ET_PAUSE:=TON.ET + ET_PAUSE;
END_IF

TON(IN:=IN AND NOT PAUSE ,PT:=SEL(TO_DINT(PT_START)-TO_DINT(ET_PAUSE)>0,T#0S,PT_START-ET_PAUSE));

Q:=TON.Q;
ET:=(ET_PAUSE+TON.ET);
IF NOT IN THEN
	ET:=T#0s;
END_IF

END_FUNCTION_BLOCK

// ---- POUs/P06_ProcessControl.TcPOU
PROGRAM P06_ProcessControl
VAR CONSTANT
	//Address constants
	HOME			:UINT:=100;
	finish			:UINT:=999;
	done			:UINT:=1000;
	
	//Robot job constants
	//Robot_Pi

END_VAR
VAR_OUTPUT
	q_bAllInHP		:BOOL;
	q_bPause		:BOOL;
END_VAR
VAR
	iStep			:UINT;
END_VAR
VAR // added by the converter: edge detectors and wires of the graphical bodies
    _rt1, _rt2, _rt3, _rt4, _rt5, _rt6, _rt7, _rt8, _rt9, _rt10, _rt11, _rt12 : R_TRIG;
    _w1 : BOOL;
END_VAR

//Select mode
IF Station.stControl.bAuto THEN
	Station.stCommand := Station.stAutoCmd;
	MEMSET(destAddr:=Station.stManCmd, fillByte:=0, n:=SIZEOF(Station.stManCmd));
ELSIF Station.stControl.bService THEN
	Station.stCommand := Station.stManCmd;
	MEMSET(destAddr:=Station.stAutoCmd, fillByte:=0, n:=SIZEOF(Station.stAutoCmd));
END_IF

//Step-sequence
CASE iStep OF
	0: //Init
	
END_CASE

//Cycle time handler
Station.tonCycleTimer(IN:=(Station.stControl.iStep >= 110 AND Station.stControl.iStep <= 240), PT:=T#10H);

//Shift handler

ACTION GeneralHP:
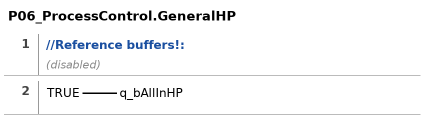
// NETWORK 1 (disabled)
// label: //Reference buffers!

// NETWORK 2
q_bAllInHP := TRUE;
END_ACTION

ACTION PartCounter:
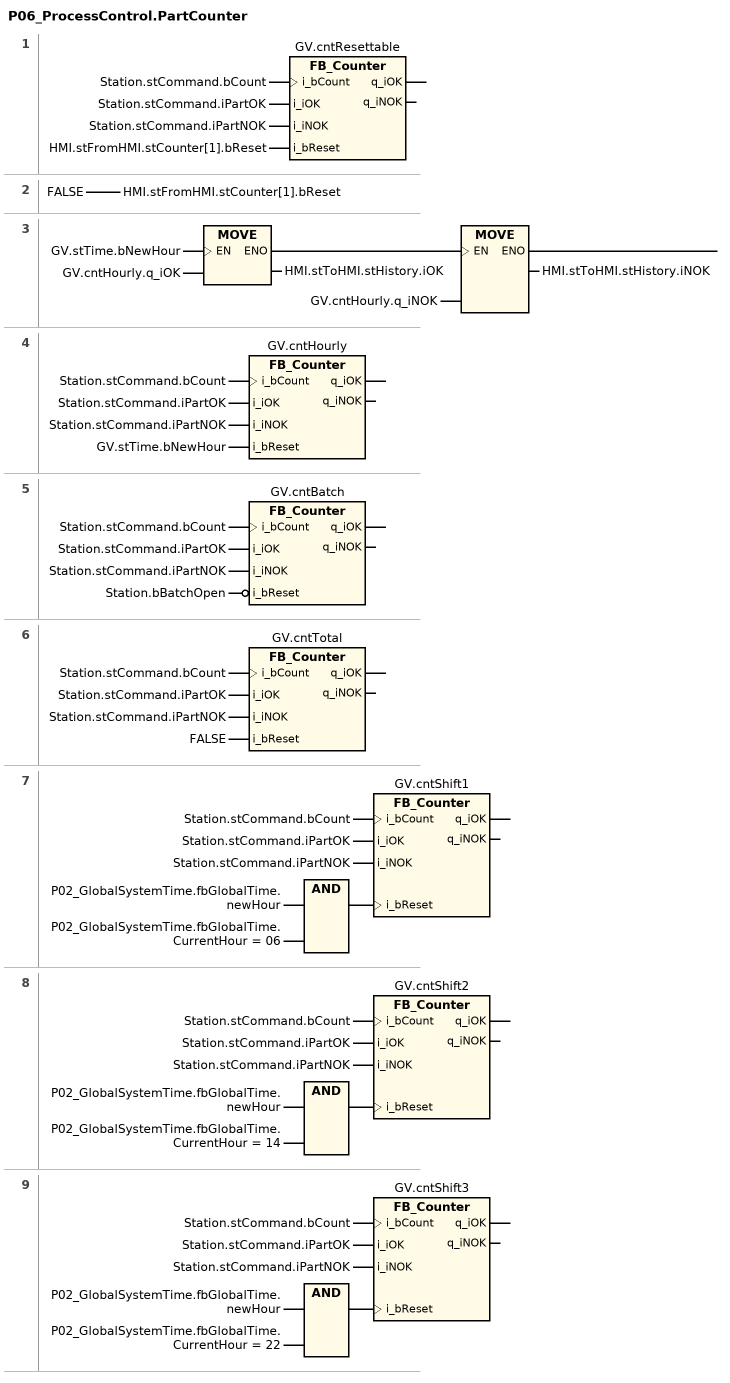
// NETWORK 1
_rt1(CLK := Station.stCommand.bCount);
GV.cntResettable(
    i_bCount := _rt1.Q,
    i_iOK := Station.stCommand.iPartOK,
    i_iNOK := Station.stCommand.iPartNOK,
    i_bReset := HMI.stFromHMI.stCounter[1].bReset); // FB_Counter

// NETWORK 2
HMI.stFromHMI.stCounter[1].bReset := FALSE;

// NETWORK 3
_rt2(CLK := GV.stTime.bNewHour);
_w1 := _rt2.Q;
IF _w1 THEN HMI.stToHMI.stHistory.iOK := GV.cntHourly.q_iOK; END_IF
_rt3(CLK := _w1);
IF _rt3.Q THEN HMI.stToHMI.stHistory.iNOK := GV.cntHourly.q_iNOK; END_IF

// NETWORK 4
_rt4(CLK := Station.stCommand.bCount);
GV.cntHourly(
    i_bCount := _rt4.Q,
    i_iOK := Station.stCommand.iPartOK,
    i_iNOK := Station.stCommand.iPartNOK,
    i_bReset := GV.stTime.bNewHour); // FB_Counter

// NETWORK 5
_rt5(CLK := Station.stCommand.bCount);
GV.cntBatch(
    i_bCount := _rt5.Q,
    i_iOK := Station.stCommand.iPartOK,
    i_iNOK := Station.stCommand.iPartNOK,
    i_bReset := NOT Station.bBatchOpen); // FB_Counter

// NETWORK 6
_rt6(CLK := Station.stCommand.bCount);
GV.cntTotal(
    i_bCount := _rt6.Q,
    i_iOK := Station.stCommand.iPartOK,
    i_iNOK := Station.stCommand.iPartNOK,
    i_bReset := FALSE); // FB_Counter

// NETWORK 7
_rt7(CLK := Station.stCommand.bCount);
_rt8(CLK := P02_GlobalSystemTime.fbGlobalTime.newHour AND (P02_GlobalSystemTime.fbGlobalTime.CurrentHour = 06));
GV.cntShift1(
    i_bCount := _rt7.Q,
    i_iOK := Station.stCommand.iPartOK,
    i_iNOK := Station.stCommand.iPartNOK,
    i_bReset := _rt8.Q); // FB_Counter

// NETWORK 8
_rt9(CLK := Station.stCommand.bCount);
_rt10(CLK := P02_GlobalSystemTime.fbGlobalTime.newHour AND (P02_GlobalSystemTime.fbGlobalTime.CurrentHour = 14));
GV.cntShift2(
    i_bCount := _rt9.Q,
    i_iOK := Station.stCommand.iPartOK,
    i_iNOK := Station.stCommand.iPartNOK,
    i_bReset := _rt10.Q); // FB_Counter

// NETWORK 9
_rt11(CLK := Station.stCommand.bCount);
_rt12(CLK := P02_GlobalSystemTime.fbGlobalTime.newHour AND (P02_GlobalSystemTime.fbGlobalTime.CurrentHour = 22));
GV.cntShift3(
    i_bCount := _rt11.Q,
    i_iOK := Station.stCommand.iPartOK,
    i_iNOK := Station.stCommand.iPartNOK,
    i_bReset := _rt12.Q); // FB_Counter
END_ACTION

ACTION Sequence:

//Control Sequence
CASE Station.stControl.iStep OF
	0: //Initialise : Status - unkonwn
	 	IF Station.stControl.bRunning THEN
		  GeneralHP();
	 	END_IF
		IF q_bAllInHP THEN
			q_bPause := TRUE;
			Station.stControl.iStep := HOME;
		END_IF
		
	
	HOME: //Home : All actuators in HP, wait for START
		Station.stControl.iStep_Prev := 0;
		q_bPause := FALSE;
		GeneralHP();
		IF Station.stControl.bRunning THEN
			Station.stControl.iStep := 110;
		END_IF
		
	110: //Start feeder
		//IF feebdack ok go 200
		
	200: //Buffer Sequence
		//Check input buffer
		IF IN.bSensor_TrayInReady THEN //OK path
			Station.stControl.iStep_Prev := Station.stControl.iStep;
			Station.stControl.iStep := 300;
		ELSE //NOK path
			Station.stControl.iStep_Prev := Station.stControl.iStep;
			Station.stControl.iStep := 210;
			;
		END_IF
	
	210: //Actuate buffer 
		//IF buffer actuation done go 220
	
	220: //Check buffer supply
		//IF buffer position 10 and NOT IN.bSensor_TrayInReady go done
		//IF buffer position <= 10 go 200
		
	300: //Convey carrier
		//IF IN.bSensor_TrayInPick and IN.bSensor_TrayInPlace go 400
		
	400://Robot start
		//In tray position ++
		//Robot job: pick up parts
		//IF Robot feedback OK go 430
		//IF Robot feecback NOK go 420
	
	420://Record missing piece in tray
		//Go to 430
	
	430://Greasing sequence
		//Robot Job := go to greasing
		//IF Robot feedback ok go to 440
	
	440://Grease 
		//IF Greaser feedback ok go 450
	
	450://Turn for greasing
		//Robot Job := turn for greasing
		//IF Robot feedback ok go 460:
	
	460://Grease
		//IF Greaser feedback ok go 500
		
	500://Push BBs to jig
		//IF feedback ok go 600
		//Have a timer for when next push is available	
	
	600://Inspect BB pick position
		//Camera Job := inspect pick BBs
		//IF Job Result OK go 700
		//IF Job Result NOK go 500
	
	700://Attatch BBs
		//Robot Job := attatch BBs
		//IF Robot feedback ok go 800
	
	800://Inspect attatched BBs
		//Camera job := inspect attatched BBs
		//IF Job OK go 900 ELSE go 810
	
	810://Discard bad pats
		//Robot job: discard bad parts
		//IF Robot feedback OK go 900
		
	900://Place done piecese in tray
		//Robot job := place parts
		//IF Robot feedback OK go 910
		
	910://
		
	finish: //Cycle finished: count parts and reset robot
		PartCounter();
		Station.stCommand.bCount := FALSE;
		//IF Robot feedback ok go 120
END_CASE
END_ACTION

END_PROGRAM

// ---- FBs/Devices/FB_Counter.TcPOU
FUNCTION_BLOCK FB_Counter
VAR_INPUT
	i_bCount		:BOOL; //Must be used with edge trigger!
	i_iOK			:USINT;
	i_iNOK			:USINT;
	i_bReset		:BOOL;
END_VAR
VAR_OUTPUT
	q_iOK			:UDINT;
	q_iNOK			:UDINT;
END_VAR
VAR
	
END_VAR

//increment
IF i_bCount THEN
	q_iOK := q_iOK + i_iOK;
ELSIF i_bCount THEN
	q_iNOK := q_iNOK + i_iNOK;
END_IF;
//reset
IF i_bReset THEN
	q_iOK := 0;
	q_iNOK := 0;
END_IF

END_FUNCTION_BLOCK

// ---- POUs/Sequences/IntakeBuffer.TcPOU
PROGRAM IntakeBuffer
VAR
	bInterlocksOK			:BOOL;
	rRealPosition			:REAL;
	rNextPosition			:REAL;
END_VAR
VAR_OUTPUT
	iStep					:UINT;
	iStepTemp				:UINT;
	iPosition				:UINT;
END_VAR

CASE iPosition OF
	0:

		rNextPosition := 2;
	1:
	
		rNextPosition := 3;
	2:

		rNextPosition := 4;
	3:

		rNextPosition := 5;
	4:

		rNextPosition := 6;
	5:

		rNextPosition := 7;
	6:
	
		rNextPosition := 8;
	7:
		rNextPosition := 9;
	8:
		
		rNextPosition := 10;
	9:
		
		rNextPosition := 11;
	10:
		
		rNextPosition := 1;
		
END_CASE

bInterlocksOK := IN.bIntakeBuffer_DriveOK AND IN.bSensor_InletDoor_Closed;

iStepTemp:=iStep;
CASE iStep OF
	0: //Hold
		IF Station.stControl.bRunning THEN
			iStep := 100;
		END_IF
		
	100: //Counting trays
		IF iPosition <= 10 AND IN.bSensor_TrayInReady THEN
			iStep := 400; //Continue
		ELSIF iPosition = 10 AND NOT IN.bSensor_TrayInReady THEN
			iStep := 200; //Buffer empty
		END_IF
	
	200: //Home buffer
		IF IN.bIntakeBuffer_Homed THEN
			iStep := 300;
		END_IF
	
	300: //Call operator and pause process (in MachineControl)
		HMI.stToHMI.iMessage := CONST.MSG_FillIntakeBuffer;
		iStep := 999;
	
		
	400: //Waiting for Robot
		
		
	500: //Waiting for conveyor
		IF Conveyor.iStep = 999 THEN
			iStep := 600;
		END_IF
		
	600: //Lowering
		IF rRealPosition = rNextPosition THEN 
			iPosition := iPosition + 1;
			iStep := 999;
		END_IF
	
	999: //finish
		iStep := 0;

END_CASE
IF NOT bInterlocksOK THEN
	iStep:=iStepTemp;
END_IF

//Control
//Station.stAutoCmd.bIntakeLift_HOME := F_StepCMP(iStep, 200, 0, 0, 0, 0, 0, 0, 0, 0, 0);
//Station.stAutoCmd.bIntakeLift_DOWN := F_StepCMP(iStep, 600, 0, 0, 0, 0, 0, 0, 0, 0, 0);

END_PROGRAM

// ---- POUs/Sequences/Conveyor.TcPOU
PROGRAM Conveyor
VAR
	bInterlocksOK	:BOOL;
END_VAR
VAR_OUTPUT
	iStep			:UINT;
	iStepTemp		:UINT;
END_VAR

bInterlocksOK := IN.bConveyorDrive_OK AND NOT IN.bSensor_TrayOutReady AND NOT IN.bPickClamped AND NOT IN.bPlaceClamped;

iStepTemp:=iStep;
CASE iStep OF
	0: //Hold
		IF Station.stControl.bRunning THEN
			iStep := 100;
		END_IF
		
	100: //Waiting for Intake Buffer
		IF IntakeBuffer.iStep = 500 THEN
			iStep := 200;
		END_IF

	200: //Drive
		IF IN.bConveyor_Drive THEN
			iStep := 300;
		END_IF
	
	300: //Driving 1
		IF IN.bSensor_TrayInPick THEN
			iStep := 310;
		END_IF
	
	310: //Driving 2
		IF NOT IN.bSensor_TrayInPick THEN
			iStep := 400;
		END_IF
	
	400: //Wait for firsst contact
		IF IN.bSensor_TrayInPick THEN
			iStep := 410;
		ELSIF IN.bSensor_TrayInPlace THEN
			iStep := 450;
		END_IF
	
	410: //Lock pick position
		;
	
	999: //finish
		iStep := 0;
END_CASE
IF NOT bInterlocksOK THEN
	iStep:=iStepTemp;
END_IF

//Control
Station.stAutoCmd.bConveyorJog := F_StepCMP(iStep, 200, 300, 0, 0, 0, 0, 0, 0, 0, 0);
//ADD Clamps control

END_PROGRAM

// ---- Functions/F_StepCMP.TcPOU
FUNCTION F_StepCMP : BOOL
VAR_INPUT
	iStep			:INT:=0;
	i1				:INT:=0;
	i2				:INT:=0;
	i3				:INT:=0;
	i4				:INT:=0;
	i5				:INT:=0;
	i6				:INT:=0;
	i7				:INT:=0;
	i8				:INT:=0;
	i9				:INT:=0;
	i10				:INT:=0;
END_VAR

F_StepCMP:=((iStep=i1) OR 
			(iStep=i2) OR 
			(iStep=i3) OR 
			(iStep=i4) OR 
			(iStep=i5) OR 
			(iStep=i6) OR 
			(iStep=i7) OR 
			(iStep=i8) OR 
			(iStep=i9) OR 
			(iStep=i10)) AND
			(iStep<>0);

END_FUNCTION

// ---- POUs/Sequences/Robot.TcPOU
PROGRAM Robot
VAR
	bInterlocksOK	:BOOL;
	i				:USINT;
END_VAR
VAR_OUTPUT
	iStep			:UINT;
	iStepTemp		:UINT;
END_VAR

bInterlocksOK := Station.stRobotControl.bInterlockOK;

iStepTemp:=iStep;
CASE iStep OF
	0: //Hold
		IF Station.stControl.bRunning THEN
			iStep := 100;
		END_IF
		
	100: //Waiting for tray
		IF IN.bSensor_TrayInPick AND IN.bSensor_TrayInPlace 
			AND IN.bPickClamped AND IN.bPlaceClamped THEN
			iStep := 200;
		END_IF
		
	200: //Go to pick tray
		Station.stAutoCmd.iRobot_JobNumber := 1;
		IF P05_DeviceControl.fbRobot.q_Args[1] THEN
			iStep := 300;
		END_IF

	300: //Gripper on
		IF IN.bRobot_Gripper = Station.stCommand.bRobot_Gripper THEN
			iStep := 400;
		END_IF
		
	400: //Go to precise place
		Station.stAutoCmd.iRobot_JobNumber := 2;
		IF P05_DeviceControl.fbRobot.q_Args[2] THEN
			iStep := 500;
		END_IF
	
	500: //Gripper off
		IF IN.bRobot_Gripper = Station.stCommand.bRobot_Gripper THEN
			iStep := 600;
		END_IF
	
	600: //Go to precise pick
		Station.stAutoCmd.iRobot_JobNumber := 3;
		IF P05_DeviceControl.fbRobot.q_Args[3] THEN
			iStep := 700;
		END_IF
	
	700: //Gripper on
		IF IN.bRobot_Gripper = Station.stCommand.bRobot_Gripper THEN
			iStep := 800;
		END_IF
		
	800: //Go to greasing
		Station.stAutoCmd.iRobot_JobNumber := 4;
		IF P05_DeviceControl.fbRobot.q_Args[4] THEN
			iStep := 900;
		END_IF
		
	900: //Grease
		IF Greaser.iStep = 999 THEN
			iStep := 1000;
		END_IF
		
	1000: //Go to greasing 2
		Station.stAutoCmd.iRobot_JobNumber := 5;
		IF P05_DeviceControl.fbRobot.q_Args[5] THEN
			iStep := 1100;
		END_IF	
		
	1100: //Grease
		IF Greaser.iStep = 999 THEN
			iStep := 1200;
		END_IF
		
	1200: //Go to BB pick
		Station.stAutoCmd.iRobot_JobNumber := 6;
		IF P05_DeviceControl.fbRobot.q_Args[6] THEN
			iStep := 1300;
		END_IF	
		
	1300: //Waiting for camera
		IF Camera.iStep = 999 THEN
			iStep := 1400;
		END_IF
		
	1400: //Check for bad parts
		IF P05_DeviceControl.fbRobot.q_Result = 2#11111110 THEN
			iStep := 1500;
		ELSE
			iStep := 1410;
		END_IF
	
	1410: //Discard bad parts
		Station.stAutoCmd.iRobot_JobNumber := 7;
		IF P05_DeviceControl.fbRobot.q_Args[7] THEN
			iStep := 1420;
		END_IF	
		
	1420: //Gripper off
		IF IN.bRobot_Gripper = Station.stCommand.bRobot_Gripper THEN
			iStep := 1500;
		END_IF
		
	1500: //Go to place tray
		Station.stAutoCmd.iRobot_JobNumber := 8;
		IF P05_DeviceControl.fbRobot.q_Args[8] THEN
			iStep := 1600;
		END_IF	
	
	1600: //Gripper off
		IF IN.bRobot_Gripper = Station.stCommand.bRobot_Gripper THEN
			iStep := 1700;
		END_IF
		
	1700: //Return to init
		Station.stAutoCmd.iRobot_JobNumber := 9;
		IF P05_DeviceControl.fbRobot.q_Args[9] THEN
			iStep := 999;
		END_IF
		
	999: //finish
		iStep := 0;
END_CASE
IF NOT bInterlocksOK THEN
	iStep:=iStepTemp;
END_IF

//Control

IF F_StepCMP(iStep, 300, 400, 700, 800, 900, 1000, 1100, 1200, 1300, 1400)
OR F_StepCMP(iStep, 1410, 0, 0, 0, 0, 0, 0, 0, 0, 0) THEN
	Station.stAutoCmd.bRobot_Gripper := 2#11111110; 
ELSIF F_StepCMP(iStep, 1420, 1500, 0, 0, 0, 0, 0, 0, 0, 0) THEN
	Station.stAutoCmd.bRobot_Gripper := P05_DeviceControl.fbRobot.q_Result;
ELSE
	Station.stAutoCmd.bRobot_Gripper := 2#00000000;
END_IF

END_PROGRAM

// ---- POUs/P05_DeviceControl.TcPOU
PROGRAM P05_DeviceControl
VAR
	fbGreasing			:FB_Greaser;
	fbCamera			:FB_Handshake;
	fbRobot				:FB_Handshake;
	fbConveyor			:FB_Device;
	fbPickClamp			:FB_Device;
	fbPlaceClamp		:FB_Device;
	fbFeeder			:FB_Device;	
	fbIntakeBuffer		:FB_Stepper;
	fbOutletBuffer		:FB_Stepper;
END_VAR
VAR // added by the converter: edge detectors and wires of the graphical bodies
    _rt1, _rt2, _rt3, _rt4, _rt5 : R_TRIG;
    _ft1, _ft2, _ft3, _ft4 : F_TRIG;
END_VAR

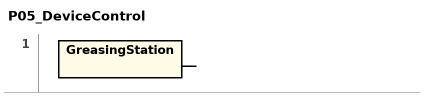
// NETWORK 1
GreasingStation();

ACTION Camera:
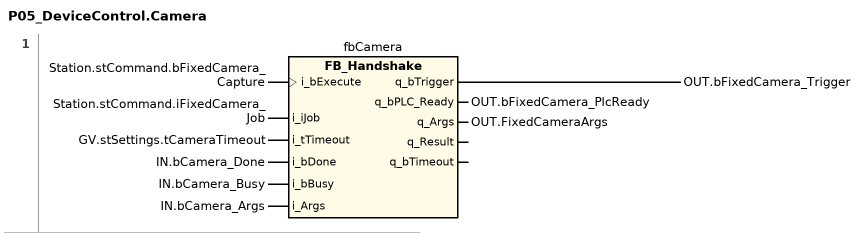
// NETWORK 1
_rt1(CLK := Station.stCommand.bFixedCamera_Capture);
fbCamera(
    i_bExecute := _rt1.Q,
    i_iJob := Station.stCommand.iFixedCamera_Job,
    i_tTimeout := GV.stSettings.tCameraTimeout,
    i_bDone := IN.bCamera_Done,
    i_bBusy := IN.bCamera_Busy,
    i_Args := IN.bCamera_Args,
    q_bPLC_Ready => OUT.bFixedCamera_PlcReady,
    q_Args => OUT.FixedCameraArgs); // FB_Handshake
OUT.bFixedCamera_Trigger := fbCamera.q_bTrigger;
END_ACTION

ACTION Conveyor:
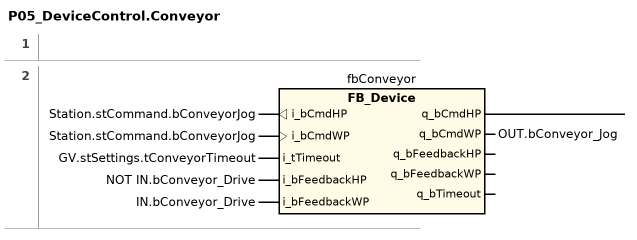
// NETWORK 1

// NETWORK 2
_ft1(CLK := Station.stCommand.bConveyorJog);
_rt2(CLK := Station.stCommand.bConveyorJog);
fbConveyor(
    i_bCmdHP := _ft1.Q,
    i_bCmdWP := _rt2.Q,
    i_tTimeout := GV.stSettings.tConveyorTimeout,
    i_bFeedbackHP := NOT IN.bConveyor_Drive,
    i_bFeedbackWP := IN.bConveyor_Drive,
    q_bCmdWP => OUT.bConveyor_Jog); // FB_Device
END_ACTION

ACTION Conveyor_PickClamp:
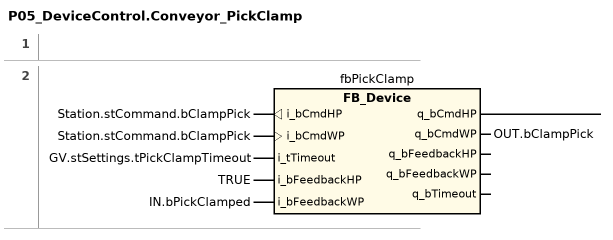
// NETWORK 1

// NETWORK 2
_ft2(CLK := Station.stCommand.bClampPick);
_rt3(CLK := Station.stCommand.bClampPick);
fbPickClamp(
    i_bCmdHP := _ft2.Q,
    i_bCmdWP := _rt3.Q,
    i_tTimeout := GV.stSettings.tPickClampTimeout,
    i_bFeedbackHP := TRUE,
    i_bFeedbackWP := IN.bPickClamped,
    q_bCmdWP => OUT.bClampPick); // FB_Device
END_ACTION

ACTION Conveyor_PlaceClamp:
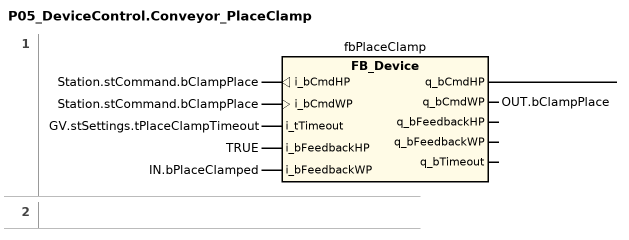
// NETWORK 1
_ft3(CLK := Station.stCommand.bClampPlace);
_rt4(CLK := Station.stCommand.bClampPlace);
fbPlaceClamp(
    i_bCmdHP := _ft3.Q,
    i_bCmdWP := _rt4.Q,
    i_tTimeout := GV.stSettings.tPlaceClampTimeout,
    i_bFeedbackHP := TRUE,
    i_bFeedbackWP := IN.bPlaceClamped,
    q_bCmdWP => OUT.bClampPlace); // FB_Device

// NETWORK 2
END_ACTION

ACTION Feeder:
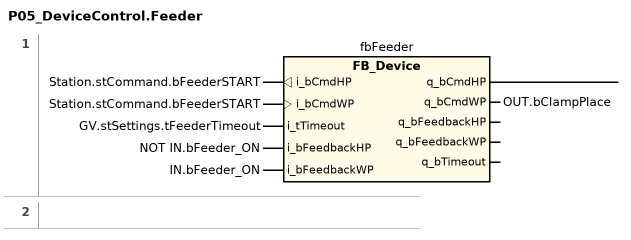
// NETWORK 1
_ft4(CLK := Station.stCommand.bFeederSTART);
_rt5(CLK := Station.stCommand.bFeederSTART);
fbFeeder(
    i_bCmdHP := _ft4.Q,
    i_bCmdWP := _rt5.Q,
    i_tTimeout := GV.stSettings.tFeederTimeout,
    i_bFeedbackHP := NOT IN.bFeeder_ON,
    i_bFeedbackWP := IN.bFeeder_ON,
    q_bCmdWP => OUT.bClampPlace); // FB_Device

// NETWORK 2
END_ACTION

ACTION GreasingStation:
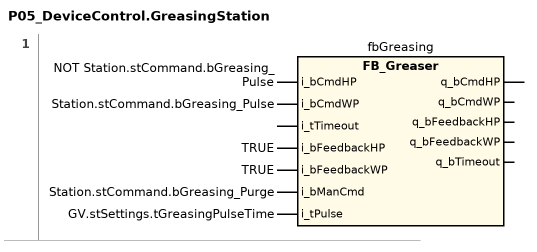
// NETWORK 1
fbGreasing(
    i_bCmdHP := NOT Station.stCommand.bGreasing_Pulse,
    i_bCmdWP := Station.stCommand.bGreasing_Pulse,
    i_bFeedbackHP := TRUE,
    i_bFeedbackWP := TRUE,
    i_bManCmd := Station.stCommand.bGreasing_Purge,
    i_tPulse := GV.stSettings.tGreasingPulseTime); // FB_Greaser
END_ACTION

ACTION IntakeBuffer:

END_ACTION

ACTION OuletBuffer:
// NETWORK 1
END_ACTION

ACTION Robot:
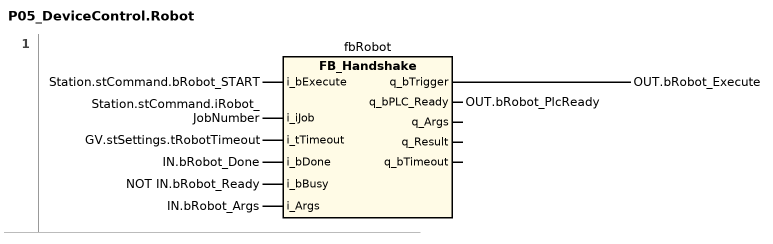
// NETWORK 1
fbRobot(
    i_bExecute := Station.stCommand.bRobot_START,
    i_iJob := Station.stCommand.iRobot_JobNumber,
    i_tTimeout := GV.stSettings.tRobotTimeout,
    i_bDone := IN.bRobot_Done,
    i_bBusy := NOT IN.bRobot_Ready,
    i_Args := IN.bRobot_Args,
    q_bPLC_Ready => OUT.bRobot_PlcReady); // FB_Handshake
OUT.bRobot_Execute := fbRobot.q_bTrigger;
END_ACTION

END_PROGRAM

// ---- FBs/Devices/FB_Greaser.TcPOU
FUNCTION_BLOCK FB_Greaser EXTENDS FB_Device
VAR_INPUT
	i_bManCmd		:BOOL; //Purge while ON, intended for manual use
	i_tPulse		:TIME; //Purge time
END_VAR
VAR_OUTPUT
END_VAR
VAR
	tPulseTimer		:TON;
END_VAR

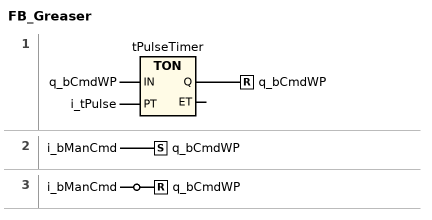
// NETWORK 1
tPulseTimer(IN := q_bCmdWP, PT := i_tPulse); // TON
q_bCmdWP R= tPulseTimer.Q;

// NETWORK 2
q_bCmdWP S= i_bManCmd;

// NETWORK 3
q_bCmdWP R= NOT i_bManCmd;

END_FUNCTION_BLOCK

// ---- FBs/Devices/FB_Device.TcPOU
FUNCTION_BLOCK FB_Device
VAR_INPUT
	i_bCmdHP				:BOOL;	//Command trigger
	i_bCmdWP				:BOOL;	//Command trigger
	i_tTimeout				:TIME;	//Time before timeout
	
	i_bFeedbackHP			:BOOL;	//Link to input, else set True
	i_bFeedbackWP			:BOOL;	//Link to input, else set True
END_VAR
VAR_OUTPUT
	q_bCmdHP				:BOOL;	//Link to output
	q_bCmdWP				:BOOL;	//Link to output
	q_bFeedbackHP			:BOOL;	//Device in HP
	q_bFeedbackWP			:BOOL;	//Device in WP
	q_bTimeout				:BOOL;	//Error
END_VAR
VAR
	tonTimeout				:TON;
END_VAR

//Go to HP
IF i_bCmdHP THEN
	q_bCmdHP := TRUE;
	q_bCmdWP := FALSE;
END_IF
//Go to WP
IF i_bCmdWP THEN
	q_bCmdWP := TRUE;
	q_bCmdHP := FALSE;
END_IF
//Do nothing if both
IF i_bCmdHP AND i_bCmdWP THEN
	q_bCmdHP := FALSE;
	q_bCmdWP := FALSE;
END_IF
//Error handler
tonTimeout(IN:=((q_bCmdHP AND NOT q_bFeedbackHP) OR (q_bCmdWP AND NOT q_bFeedbackWP)) AND NOT (i_bCmdHP OR i_bCmdWP) , PT:=i_tTimeout);
q_bTimeout := tonTimeout.Q;
//Feedback
q_bFeedbackHP := i_bFeedbackHP AND q_bCmdHP;
q_bFeedbackWP := i_bFeedbackWP AND q_bCmdWP;

END_FUNCTION_BLOCK

// ---- FBs/Devices/FB_Handshake.TcPOU
FUNCTION_BLOCK FB_Handshake
VAR_INPUT
	i_bExecute			:BOOL;						//Input
	i_iJob				:USINT;						//Job number (if only one job leave at 0)
	i_tTimeout			:TIME;

	i_bDone				:BOOL;						//Job done
	i_bBusy				:BOOL;						//Device busy
	i_Args				:BYTE;						//Device arguments
END_VAR
VAR_OUTPUT
	q_bTrigger			:BOOL;						//Activate job
	q_bPLC_Ready		:BOOL := FALSE;				//Handshake initiated
	q_Args				:ARRAY [0..9] OF BOOL;		//Information for device
	
	q_Result			:BYTE;		//Adjust for possible results
	q_bTimeout			:BOOL;
END_VAR
VAR
	i		:USINT;
	tonTimeout	:TON;
END_VAR

//Wait for device ready
IF i_bBusy THEN
	q_bTrigger := FALSE;
END_IF
//Init handshake:
IF i_bExecute AND NOT q_bPLC_Ready THEN
	q_bPLC_Ready := TRUE;
	q_bTrigger := TRUE;
	MEMSET(destAddr:=ADR(q_Args), fillByte:=0, n:=SIZEOF(q_Args));
	CASE i_iJob OF
		0:
			;
		1:
			q_Args[0] := TRUE;
		2:
			q_Args[1] := TRUE;
		3:
			q_Args[2] := TRUE;
		4:
			q_Args[3] := TRUE;
		5:
			q_Args[4] := TRUE;
		6:
			q_Args[5] := TRUE;
		7:
			q_Args[6] := TRUE;
		8:
			q_Args[7] := TRUE;
		9:
			q_Args[8] := TRUE;
		10:
			q_Args[9] := TRUE;
	END_CASE
END_IF
//Device response:
IF q_bPLC_Ready THEN
	MEMSET(destAddr:=ADR(q_Result), fillByte:=0, n:=SIZEOF(q_Result));
	IF i_bDone THEN 
		q_Result := i_Args;
		q_bPLC_Ready := FALSE;
	END_IF
END_IF
//Timeout
tonTimeout(IN:=q_bPLC_Ready, PT:=i_tTimeout);
IF tonTimeout.Q THEN
	q_bPLC_Ready := FALSE;
END_IF
q_bTimeout := tonTimeout.Q;

END_FUNCTION_BLOCK

// ---- FBs/Devices/FB_Stepper.TcPOU
FUNCTION_BLOCK FB_Stepper EXTENDS FB_Device
VAR_INPUT	
END_VAR
VAR_OUTPUT
END_VAR
VAR
END_VAR

//Add the tc2_mc function blocks here

END_FUNCTION_BLOCK

// ---- POUs/Sequences/Greaser.TcPOU
PROGRAM Greaser
VAR
	bInterlocksOK	:BOOL;
	tonGreasingTime	:TON;
END_VAR
VAR_OUTPUT
	iStep			:UINT;
	iStepTemp		:UINT;
END_VAR

bInterlocksOK := IN.bGreasing_LevelOK AND IN.bGreasing_PressureOK;

tonGreasingTime(IN:=(iStep=200), PT:=T#500MS);

iStepTemp:=iStep;
CASE iStep OF
	0: //Hold
		IF Station.stControl.bRunning THEN
			iStep := 100;
		END_IF
		
	100: //Waiting for robot
		IF Robot.iStep = 900 OR Robot.iStep = 1100 THEN
			iStep := 200;
		END_IF

	200: //Pulse
		IF tonGreasingTime.Q THEN
			iStep := 999;
		END_IF

	999: //finish
		iStep := 0;
END_CASE
IF NOT bInterlocksOK THEN
	iStep:=iStepTemp;
END_IF

//Control
Station.stAutoCmd.bGreasing_Pulse := F_StepCMP(iStep, 200, 0, 0, 0, 0, 0, 0, 0, 0, 0);

END_PROGRAM

// ---- POUs/Sequences/Camera.TcPOU
PROGRAM Camera
VAR
	bInterlocksOK	:BOOL;
END_VAR
VAR_OUTPUT
	iStep			:UINT;
	iStepTemp		:UINT;
END_VAR

bInterlocksOK := IN.bCamera_On;

iStepTemp:=iStep;
CASE iStep OF
	0: //Hold
		IF Station.stControl.bRunning THEN
			iStep := 100;
		END_IF
		
	100: //Waiting for Robot
		IF Robot.iStep = 1300 THEN
			iStep := 200;
		END_IF

	200: //Inspect BBs
		Station.stAutoCmd.iFixedCamera_Job := 1;
		IF P05_DeviceControl.fbCamera.q_Args[1] THEN
			iStep := 999;
		END_IF
	
	999: //finish
		iStep := 0;
END_CASE
IF NOT bInterlocksOK THEN
	iStep:=iStepTemp;
END_IF

//Control
IF F_StepCMP(iStep, 200, 0, 0, 0, 0, 0, 0, 0, 0, 0) THEN
	Station.stAutoCmd.iFixedCamera_Job := 1;
ELSE
	Station.stAutoCmd.iFixedCamera_Job := 0;
END_IF

END_PROGRAM

// ---- POUs/P99_HMIControl.TcPOU
PROGRAM P99_HMIControl
VAR
	i:UDINT;
	j:UDINT;
END_VAR

//----------------Header---------------------//
IF Station.stControl.bAuto THEN
	HMI.stToHMI.stHeader.bControlMode := 0;
ELSIF Station.stControl.bService THEN
	HMI.stToHMI.stHeader.bControlMode := 1;
END_IF

IF Station.stControl.bStopping THEN
	HMI.stToHMI.stHeader.iStatus := 0;
ELSIF Station.stControl.bStopped THEN
	HMI.stToHMI.stHeader.iStatus := 1;
ELSIF Station.stControl.bStarting THEN
	HMI.stToHMI.stHeader.iStatus := 2;
ELSIF Station.stControl.bRunning THEN
	HMI.stToHMI.stHeader.iStatus := 3;
ELSIF Station.stControl.bPaused THEN
	HMI.stToHMI.stHeader.iStatus := 4;
END_IF

HMI.stToHMI.stHeader.sCycleTime := F_TimerToString(Station.tonCycleTimer.ET);
HMI.stToHMI.stHeader.sDate := GV.stTime.sDate;
HMI.stToHMI.stHeader.sTime := GV.stTime.sTime;

IF Station.bBatchOpen THEN
	HMI.stToHMI.stHeader.sBatch := Station.stBatch.sBatchNumber;
ELSE
	HMI.stToHMI.stHeader.sBatch := '-';
END_IF

//------------------Footer---------------------//
//Footer commands:
HMI.stToHMI.stFooter.bAuto_Enable := TRUE;
HMI.stToHMI.stFooter.bService_Enable := NOT Station.stControl.bRunning;
HMI.stToHMI.stFooter.bStart_Enable := Station.stControl.bStartConditionsOK;
HMI.stToHMI.stFooter.bStop_Enable := TRUE;
HMI.stToHMI.stFooter.bPause_Enable := TRUE;
//Footer feedback:
HMI.stToHMI.stFooter.bAuto := Station.stControl.bAuto;
HMI.stToHMI.stFooter.bService := Station.stControl.bService;
HMI.stToHMI.stFooter.bStart := Station.stControl.bRunning OR (Station.stControl.bStarting AND GV.stTime.bClock_500ms);
HMI.stToHMI.stFooter.bPause := Station.stControl.bPaused;
HMI.stToHMI.stFooter.bStop := Station.stControl.bStopped OR (Station.stControl.bStopping AND GV.stTime.bClock_500ms);

//---------------------------------------------PnID---------------------------------------//

//----------------Robot--------------------//
//Robot controller:
HMI.stToHMI.stRobot.bPowerOn := Station.stRobotControl.bPoweredOn OR (Station.stRobotControl.bStarting AND GV.stTime.bClock_500ms);
HMI.stToHMI.stRobot.bPowerOff := Station.stRobotControl.bPoweredOff OR (Station.stRobotControl.bStopping AND GV.stTime.bClock_500ms);
HMI.stToHMI.stRobot.bInit := Station.stRobotControl.bInit AND GV.stTime.bClock_500ms;
HMI.stToHMI.stRobot.bStart := Station.stRobotControl.bRunning;
HMI.stToHMI.stRobot.bStop := Station.stRobotControl.bStopped;
HMI.stToHMI.stRobot.bPause := Station.stRobotControl.bPaused;
//Robot station:
HMI.stRobot.bInterlocksOK := Station.stRobotControl.bInterlockOK;
HMI.stRobot.iStep := Station.stRobotControl.iStep;
IF Station.stCommand.iRobot_JobNumber = 0 THEN
	HMI.stRobot.iStatus := 0;
ELSE //if not error and not step waiting
	HMI.stRobot.iStatus := 3;
END_IF
//HMI.stToHMI.stRobot.sStatus := Device.status

//--------------Lifts----------------------//
//Intake lift (left)
//Service mode commands
IF HMI.stFromHMI.stLiftIntake.bHome AND Station.stControl.bService THEN
	Station.stManCmd.bIntakeLift_HOME := TRUE;
END_IF
IF Station.stControl.bService THEN
	Station.stManCmd.iIntakeLift_SP := HMI.stFromHMI.stLiftIntake.iPosition;
END_IF
//Visualisation
HMI.stToHMI.stLiftIntake.bHome := Station.stManCmd.bIntakeLift_HOME AND GV.stTime.bClock_500ms;
IF HMI.stToHMI.stLiftIntake.iPosition > 10 THEN
	HMI.stToHMI.stLiftIntake.iPosition := 10;
END_IF
IF HMI.stToHMI.stLiftIntake.iPosition <1 THEN
	HMI.stToHMI.stLiftIntake.iPosition := 1;
END_IF

//Outlet lift (right)
//Service mode commands
IF HMI.stFromHMI.stLiftOutlet.bHome AND Station.stControl.bService THEN
	Station.stManCmd.bOutletLift_HOME := TRUE;
END_IF
IF Station.stControl.bService THEN
	Station.stManCmd.iOutletLift_SP := HMI.stFromHMI.stLiftOutlet.iPosition;
END_IF
//Visualisation
HMI.stToHMI.stLiftOutlet.bHome := Station.stManCmd.bOutletLift_HOME AND GV.stTime.bClock_500ms;
IF HMI.stToHMI.stLiftOutlet.iPosition > 10 THEN
	HMI.stToHMI.stLiftOutlet.iPosition := 10;
END_IF
IF HMI.stToHMI.stLiftOutlet.iPosition <1 THEN
	HMI.stToHMI.stLiftOutlet.iPosition := 1;
END_IF

//--------------Conveyor----------------------//
HMI.stToHMI.stPID.bConveyor_Moving := IN.bConveyor_Drive;
Station.stManCmd.bConveyorJog := HMI.stFromHMI.bConveyorJog; //Service mode command

//---------------Cameras---------------------//
//Robot camera (above)
HMI.stToHMI.stRobotCamera.bCapturing := Station.stCommand.bRobotCamera_Capture;
(*
IF Device.Pass THEN
	HMI.stToHMI.stRobotCamera.sJobResult := 'Pass';
ELSIF Device.Fail THEN
	HMI.stToHMI.stRobotCamera.sJobResult := 'Fail';
ELSE
	HMI.stToHMI.stRobotCamera.sJobResult := '';
END_IF
*)
//HMI.stToHMI.stRobotCamera.sCameraStatus := Device.status

//Fixed camera (above)
HMI.stToHMI.stFixedCamera.bCapturing := Station.stCommand.bFixedCamera_Capture;
HMI.stCamera.bInterlocksOK := IN.bCamera_On;
(*
IF Device.Pass THEN
	HMI.stToHMI.stFixedCamera.sJobResult := 'Pass';
ELSIF Device.Fail THEN
	HMI.stToHMI.stFixedCamera.sJobResult := 'Fail';
ELSE
	HMI.stToHMI.stFixedCamera.sJobResult := '';
END_IF
*)
//HMI.stToHMI.stFixedCamera.sCameraStatus := Device.status

//----------------Greasing station----------//
//Service mode commands
Station.stManCmd.tGreasing_Time := UINT_TO_TIME(HMI.stFromHMI.stGreasing.iTime);
Station.stManCmd.bGreasing_Pulse := HMI.stFromHMI.stGreasing.bPulse;
Station.stManCmd.bGreasing_Purge := HMI.stFromHMI.stGreasing.bPurge;
HMI.stGreasing.bInterlocksOK := TRUE;

//-----------------Feeder--------------------//
IF HMI.stFromHMI.stFeeder.bActivate THEN
	Station.stManCmd.bFeederSTART := TRUE;
ELSIF HMI.stFromHMI.stFeeder.bDeactivate THEN
	Station.stManCmd.bFeederSTART := FALSE;
END_IF

HMI.stToHMI.stFeeder.bActivate := IN.bFeeder_ON;
HMI.stToHMI.stFeeder.bDeactivate := NOT IN.bFeeder_ON;

//---------------LastTray-------------------//
IF HMI.stFromHMI.iSelectedTray < 1 THEN
	HMI.stFromHMI.iSelectedTray := 1;
END_IF
IF HMI.stFromHMI.iSelectedTray >10 THEN
	HMI.stFromHMI.iSelectedTray := 10;
END_IF
HMI.stLastTray := GV.aTrays[HMI.stFromHMI.iSelectedTray];

//----------------Sensors------------------//
HMI.stToHMI.stPID.bTray_Ready_Left := IN.bSensor_TrayInReady;
HMI.stToHMI.stPID.bTray_Ready_Right := IN.bSensor_TrayOutReady;
HMI.stToHMI.stPID.bTray_PickPosition := IN.bSensor_TrayInPick;
HMI.stToHMI.stPID.bTray_PlacePosition := IN.bSensor_TrayInPlace;

//---------------POP-ups--------------------//
IF HMI.iMenu <> 0 THEN
	HMI.iPopupMenu := 0;
END_IF

//---------------------------------------BATCH page----------------------------------------//

HMI.stToHMI.stBatch.bBatchOpen := Station.bBatchOpen;
HMI.stToHMI.stBatch.bBatchClose := Station.bBatchClosed;

//--------------------------------------PRODUCTIVITY page----------------------------------//
//Resettable counter:
HMI.stToHMI.stCounter[1].iOK := GV.cntResettable.q_iOK;
HMI.stToHMI.stCounter[1].iNOK := GV.cntResettable.q_iNOK;
//Hurly counter
HMI.stToHMI.stCounter[2].iOK := GV.cntHourly.q_iOK;
HMI.stToHMI.stCounter[2].iNOK := GV.cntHourly.q_iNOK;
//Batch counter
HMI.stToHMI.stCounter[3].iOK := GV.cntBatch.q_iOK;
HMI.stToHMI.stCounter[3].iNOK := GV.cntBatch.q_iNOK;
//Total counter
HMI.stToHMI.stCounter[4].iOK := GV.cntTotal.q_iOK;
HMI.stToHMI.stCounter[4].iNOK := GV.cntTotal.q_iNOK;
//Trend 
HMI.stToHMI.stHistory.bShift1 := GV.stTime.CurrentHour >= 6 AND GV.stTime.CurrentHour <14;
HMI.stToHMI.stHistory.bShift2 := GV.stTime.CurrentHour >= 14 AND GV.stTime.CurrentHour <22;
HMI.stToHMI.stHistory.bShift3 := GV.stTime.CurrentHour >= 22 OR GV.stTime.CurrentHour <6;

END_PROGRAM

// ---- Functions/F_TimerToString.TcPOU
FUNCTION F_TimerToString : STRING
VAR_INPUT
	i_tTime				:TIME;
END_VAR
VAR
	iTimeInSec			:UDINT;
	iHours				:UDINT;
	iMinutes			:UDINT;
	iSeconds			:UDINT;
	sQuery				:STRING;
END_VAR

iTimeInSec:=TO_UDINT(i_tTIme)/1000;

iHours:=iTimeInSec/3600;
iMinutes:=(iTimeInSec/60)-(iHours*60);
iSeconds:=iTimeInSec - (iMinutes*60) - (iHours*3600);
(*
IF iHours = 0 THEN
	sQuery:='00:';
ELSIF iHours > 0 AND iHours < 10 THEN
	sQuery:=CONCAT('0',TO_STRING(iHours));
	sQuery:=CONCAT(sQuery,':');
ELSE
	sQuery:=TO_STRING(iHours);
	sQuery:=CONCAT(sQuery,':');
END_IF
*)
IF iMinutes = 0 THEN
	sQuery:='00:';
ELSIF iMinutes > 0 AND iMinutes < 10 THEN
	sQuery:=CONCAT('0',TO_STRING(iMinutes));
	sQuery:=CONCAT(sQuery,':');
ELSE
	sQuery:=TO_STRING(iMinutes);
	sQuery:=CONCAT(sQuery,':');
END_IF

IF iSeconds = 0 THEN
	sQuery:=CONCAT(sQuery,'00');
ELSIF iSeconds > 0 AND iSeconds < 10 THEN
	sQuery:=CONCAT(sQuery,'0');
	sQuery:=CONCAT(sQuery,TO_STRING(iSeconds));
ELSE
	sQuery:=CONCAT(sQuery,TO_STRING(iSeconds));
END_IF


F_TimerToString:=sQuery;

END_FUNCTION

// ---- POUs/Simulation/Service_sim.TcPOU
PROGRAM Service_sim
//---------------------------------Acutators simulation----------------------------------//
VAR
	TON_0: TON;
	TON_1: TON;
	TON_2: TON;
	TON_3: TON;
	TON_4: TON;
END_VAR

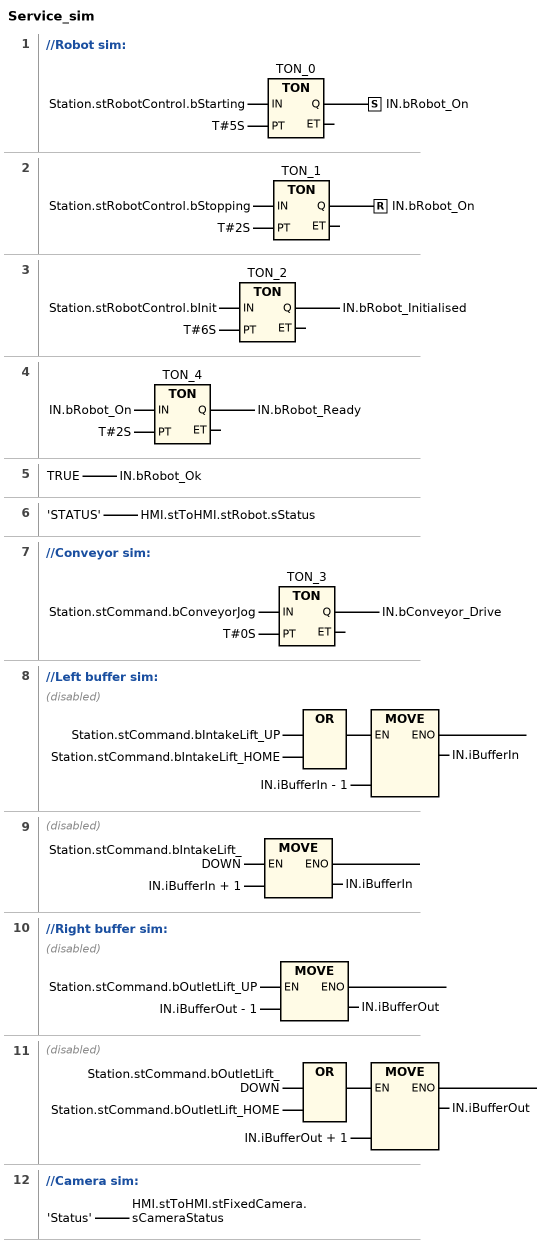
// NETWORK 1
// label: //Robot sim
TON_0(IN := Station.stRobotControl.bStarting, PT := T#5S); // TON
IN.bRobot_On S= TON_0.Q;

// NETWORK 2
TON_1(IN := Station.stRobotControl.bStopping, PT := T#2S); // TON
IN.bRobot_On R= TON_1.Q;

// NETWORK 3
TON_2(IN := Station.stRobotControl.bInit, PT := T#6S); // TON
IN.bRobot_Initialised := TON_2.Q;

// NETWORK 4
TON_4(IN := IN.bRobot_On, PT := T#2S); // TON
IN.bRobot_Ready := TON_4.Q;

// NETWORK 5
IN.bRobot_Ok := TRUE;

// NETWORK 6
HMI.stToHMI.stRobot.sStatus := 'STATUS';

// NETWORK 7
// label: //Conveyor sim
TON_3(IN := Station.stCommand.bConveyorJog, PT := T#0S); // TON
IN.bConveyor_Drive := TON_3.Q;

// NETWORK 8 (disabled)
// label: //Left buffer sim
// IF Station.stCommand.bIntakeLift_UP OR Station.stCommand.bIntakeLift_HOME THEN
//     IN.iBufferIn := IN.iBufferIn - 1;
// END_IF

// NETWORK 9 (disabled)
// IF Station.stCommand.bIntakeLift_DOWN THEN IN.iBufferIn := IN.iBufferIn + 1; END_IF

// NETWORK 10 (disabled)
// label: //Right buffer sim
// IF Station.stCommand.bOutletLift_UP THEN IN.iBufferOut := IN.iBufferOut - 1; END_IF

// NETWORK 11 (disabled)
// IF Station.stCommand.bOutletLift_DOWN OR Station.stCommand.bOutletLift_HOME THEN
//     IN.iBufferOut := IN.iBufferOut + 1;
// END_IF

// NETWORK 12
// label: //Camera sim
HMI.stToHMI.stFixedCamera.sCameraStatus := 'Status';

END_PROGRAM

// ---- POUs/Sequences/Feeder.TcPOU
PROGRAM Feeder
VAR
	bInterlocksOK	:BOOL;
END_VAR
VAR_OUTPUT
	iStep			:UINT;
	iStepTemp		:UINT;
END_VAR

bInterlocksOK := Robot.iStep <> 1200;

iStepTemp:=iStep;
CASE iStep OF
	0: //Hold
		IF Station.stControl.bRunning THEN
			iStep := 100;
		END_IF
		
	100: //Work
		;
END_CASE
IF NOT bInterlocksOK THEN
	iStep:=iStepTemp;
END_IF

//Control
Station.stAutoCmd.bFeederSTART := F_StepCMP(iStep, 100, 0, 0, 0, 0, 0, 0, 0, 0, 0);

END_PROGRAM

// ---- FBs/FB_AlarmDiagnostic.TcPOU
FUNCTION_BLOCK FB_AlarmDiagnostic
VAR_INPUT
	i_bEnable				:BOOL:=TRUE;
	i_iID					:INT;
	i_bInput				:BOOL;
	i_iOnDelay				:DINT:=0;
	i_bReset				:BOOL;
	i_bTest					:BOOL;
	i_bActive				:BOOL;
	i_sDisplayText			:STRING:='';
END_VAR
VAR_OUTPUT
	q_bActive				:BOOL;
	q_iDetections			:INT;
END_VAR
VAR
	TON						:TON;
END_VAR
VAR // added by the converter: edge detectors and wires of the graphical bodies
    _rt1 : R_TRIG;
    _w1 : BOOL;
END_VAR

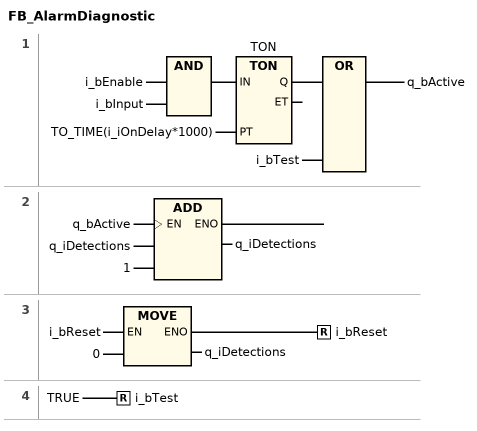
// NETWORK 1
TON(IN := i_bEnable AND i_bInput, PT := TO_TIME(i_iOnDelay*1000));
q_bActive := TON.Q OR i_bTest;

// NETWORK 2
_rt1(CLK := q_bActive);
IF _rt1.Q THEN q_iDetections := q_iDetections + 1; END_IF

// NETWORK 3
_w1 := i_bReset;
IF _w1 THEN q_iDetections := 0; END_IF
i_bReset R= _w1;

// NETWORK 4
i_bTest R= TRUE;

END_FUNCTION_BLOCK

// ---- Functions/F_Message.TcPOU
FUNCTION F_Message : BOOL
VAR_INPUT
	iMessageIndex		:UINT;
	sSeverity			:STRING; //error, warning or message
END_VAR
VAR
END_VAR

IF sSeverity = 'error' THEN //Highest priority, overwrite everything
	HMI.stToHMI.iMessageSeverity := 100; 
	HMI.stToHMI.iMessage := iMessageIndex;
END_IF

IF sSeverity = 'warning' AND HMI.stToHMI.iMessageSeverity < 50 THEN //Priority 50, overwrite everything else
	HMI.stToHMI.iMessageSeverity := 50;
	HMI.stToHMI.iMessage := iMessageIndex;
END_IF

IF sSeverity = 'message' AND HMI.stToHMI.iMessageSeverity < 10 THEN //Priority 10, overwrite everything else
	HMI.stToHMI.iMessageSeverity := 10;
	HMI.stToHMI.iMessage := iMessageIndex;
END_IF

//Reset message
IF iMessageIndex = 0 THEN
	HMI.stToHMI.iMessage := 0;
	HMI.stToHMI.iMessageSeverity := 0;
END_IF

END_FUNCTION

// ---- POUs/P00_Mapping.TcPOU
PROGRAM P00_Mapping
VAR
END_VAR

END_PROGRAM

// ---- POUs/P01_AnalogScaling.TcPOU
PROGRAM P01_AnalogScaling
VAR
END_VAR

// NETWORK 1

END_PROGRAM

// ---- POUs/Sequences/OutletBuffer.TcPOU
PROGRAM OutletBuffer
VAR
	bInterlocksOK	:BOOL;
	iPosition		:UINT;
	rNextPosition	:REAL;
END_VAR
VAR_OUTPUT
	iStep			:UINT;
	iStepTemp		:UINT;
END_VAR
VAR_INPUT
	rRealPosition	:REAL;
END_VAR

CASE iPosition OF
	0:

		rNextPosition := 10;
	1:
	
		rNextPosition := 9;
	2:

		rNextPosition := 8;
	3:

		rNextPosition := 7;
	4:

		rNextPosition := 6;
	5:

		rNextPosition := 5;
	6:
	
		rNextPosition := 4;
	7:
		rNextPosition := 3;
	8:
		
		rNextPosition := 2;
	9:
		
		rNextPosition := 1;
	10:
		
		rNextPosition := 10;
		
END_CASE

bInterlocksOK := IN.bOutletBuffer_DriveOK AND IN.bSensor_OutletDoor_Closed;

iStepTemp:=iStep;
CASE iStep OF
	0: //Hold
		IF Station.stControl.bRunning THEN
			iStep := 100;
		END_IF
		
	100: //Waiting for conveyor
		IF Conveyor.iStep = 999 AND IN.bSensor_TrayOutReady THEN
			iStep := 200;
		END_IF
		
	200: //Move UP
		IF rRealPosition = rNextPosition THEN
			iPosition := iPosition + 1;
			iStep := 300;
		END_IF
		
	300: //Check if homing required
	 	IF IN.bIntakeBuffer_Homed THEN
			iStep := 400;
		ELSE
			iStep := 999;
		END_IF
		
	400: //Homing
		IF IN.bOutletBuffer_Homed THEN
			iStep := 999;
		END_IF
		
	999: //finish
		iStep := 0;

END_CASE
IF NOT bInterlocksOK THEN
	iStep:=iStepTemp;
END_IF

//Control
Station.stAutoCmd.bIntakeLift_HOME := F_StepCMP(iStep, 400, 0, 0, 0, 0, 0, 0, 0, 0, 0);
Station.stAutoCmd.bOutletLift_UP := F_StepCMP(iStep, 200, 0, 0, 0, 0, 0, 0, 0, 0, 0);

END_PROGRAM

// ---- POUs/Simulation/Simulation.TcPOU
PROGRAM Simulation
VAR
	Lift1	:TON;
END_VAR

//Intake lift simulation:
IF HMI.stFromHMI.stLiftIntake.bGoUp THEN
	
	HMI.stFromHMI.stLiftIntake.bGoUp := FALSE;
END_IF

END_PROGRAM
